// TwinCAT 3 PLC project Fraktal_Core
// Title: Fraktal_Core
// Company: fraktal-automation
// Author: fraktal-automation
// ProjectVersion: 0.25.0.0
// Description: Fraktal Core framework library: contracts, base classes (CM/EM/Unit), PermIntlk, profiler, connector base, recipe provider (Core 2.2).
// ProgramVersion: 3.1.4026.24
// libraries:
//   Tc2_Standard, * (Beckhoff Automation GmbH)
//   Tc2_EtherCAT, * (Beckhoff Automation GmbH)
//   Tc2_System, * (Beckhoff Automation GmbH)
//   Tc2_Utilities, * (Beckhoff Automation GmbH)
//   Tc3_Module, * (Beckhoff Automation GmbH)
//   Tc3_IPCDiag, * (Beckhoff Automation GmbH)
// project tree:
//   Connectivity/ FB_LineDataV3.TcPOU, FB_ShiftSchedule.TcPOU, FB_ConfigSnapshot.TcPOU, F_AppendTopologyConfig.TcPOU, FB_AsciiLink.TcPOU, FB_DeviceConnectorBase.TcPOU, FB_EcBusHealth.TcPOU, FB_EcFieldbusScanner.TcPOU, FB_IoTopologyPublisher.TcPOU, FB_LocalAccessProvider.TcPOU, FB_ConfigSetDocument.TcPOU, FB_MediumConfigStore.TcPOU, FB_PersistMediumBase.TcPOU, FB_RetainPersistMedium.TcPOU, FB_LocalPartCarrier.TcPOU (not stored), FB_LocalRecipeProvider.TcPOU, FB_LocalConfigStore.TcPOU, FB_PersistentDataWriter.TcPOU, FB_SimByteChannel.TcPOU (not stored), FB_TcpChannelTc3.TcPOU (not stored), FB_LineData.TcPOU, FB_LineLocalSource.TcPOU, FB_LineAdsSource.TcPOU
//   DUTs/ ST_ShiftRecordV3.TcDUT, ST_ShiftCalendarV3.TcDUT, ST_ShiftRowV3.TcDUT, ST_ShiftCalendarV2.TcDUT, ST_ShiftRowV2.TcDUT, ST_ConfigFeatures.TcDUT, ST_LocalRecipeCatalog.TcDUT, ST_LocalRecipeRecord.TcDUT, E_AccessLevel.TcDUT (not stored), E_AlarmState.TcDUT (not stored), E_AsciiLinkEvent.TcDUT, E_ByteChannelState.TcDUT (not stored), E_CarrierKind.TcDUT (not stored), E_Category.TcDUT (not stored), E_ChannelDir.TcDUT (not stored), E_ChannelKind.TcDUT (not stored), E_ExecState.TcDUT (not stored), E_FieldbusLossReaction.TcDUT (not stored), E_GatedAction.TcDUT, E_HbResult.TcDUT (not stored), E_HostEventKind.TcDUT, E_LinkReaction.TcDUT (not stored), E_MachineState.TcDUT (not stored), E_Mode.TcDUT (not stored), E_ModeSwitchShield.TcDUT (not stored), E_PowerGroupKind.TcDUT (not stored), E_PowerState.TcDUT (not stored), E_SafetyDeviceKind.TcDUT (not stored), E_SafetyState.TcDUT (not stored), E_ModeSwitchStyle.TcDUT (not stored), E_ModuleType.TcDUT (not stored), E_NodeState.TcDUT (not stored), E_Reason.TcDUT, E_RecipeSource.TcDUT (not stored), E_ReleaseKind.TcDUT (not stored), E_ResetClass.TcDUT (not stored), E_RunStyle.TcDUT (not stored), E_Severity.TcDUT (not stored), E_StepResult.TcDUT (not stored), E_TimeClass.TcDUT (not stored), E_Verdict.TcDUT (not stored), ST_AccessPolicy.TcDUT, ST_AlarmEvent.TcDUT, ST_AlarmMeta.TcDUT, ST_BusNode.TcDUT, ST_CommandInfo.TcDUT, E_CommandStyle.TcDUT, ST_ManualEnableStatus.TcDUT, ST_CondRecord.TcDUT (not stored), ST_CycleProfile.TcDUT, ST_CycleSummary.TcDUT, ST_DecisionRequest.TcDUT (not stored), ST_Diagnostic.TcDUT, ST_EngineeringGate.TcDUT, ST_FieldbusTopology.TcDUT, E_HmiRequestKind.TcDUT, E_ConfigKind.TcDUT, E_ConfigRestorePolicy.TcDUT, E_ConfigStore.TcDUT, E_ConfigValueType.TcDUT, E_EngUnit.TcDUT, ST_ConfigPersistStatus.TcDUT, ST_ConfigRecord.TcDUT, ST_ConfigSetInfo.TcDUT, ST_HmiRequest.TcDUT (not stored), E_ConfigStorage.TcDUT, E_LineRole.TcDUT, ST_LineDataParCfg.TcDUT, ST_LineDataParCmd.TcDUT, ST_LineDataOutCmd.TcDUT, ST_ShiftCalendar.TcDUT, ST_ShiftRecord.TcDUT, ST_LineRecord.TcDUT, ST_LineImage.TcDUT, ST_LineStatus.TcDUT, ST_ConfigAccess.TcDUT, ST_DataClassPolicy.TcDUT, ST_ConfigWriteDef.TcDUT, ST_ConfigEntry.TcDUT, ST_ConfigPage.TcDUT (not stored), ST_HmiResponse.TcDUT, ST_HostEvent.TcDUT, ST_IntlkCond.TcDUT (not stored), ST_IoChannel.TcDUT, ST_IoPointIdentity.TcDUT (not stored), ST_MeasRecord.TcDUT (not stored), ST_ModePolicy.TcDUT (not stored), ST_ModelField.TcDUT (not stored), ST_ModelId.TcDUT (not stored), ST_ModuleStatus.TcDUT, ST_ControlDomainStatus.TcDUT (not stored), ST_ControlPowerStatus.TcDUT (not stored), ST_PowerGroupStatus.TcDUT (not stored), ST_SafetyDeviceStatus.TcDUT (not stored), ST_SafetyStatus.TcDUT (not stored), ST_ModuleTiming.TcDUT (not stored), ST_Nameplate.TcDUT (not stored), ST_Oee.TcDUT (not stored), ST_OeeSample.TcDUT (not stored), ST_PartContext.TcDUT (not stored), ST_PartResult.TcDUT, ST_ReleaseReason.TcDUT (not stored), ST_ReleaseReport.TcDUT (not stored), ST_StepRecord.TcDUT, ST_StateFlag.TcDUT, ST_SequenceStepDef.TcDUT, ST_SequenceCursor.TcDUT, ST_SequenceAnnotation.TcDUT, ST_SequenceStep.TcDUT, ST_StepTiming.TcDUT, ST_SignalTowerOut.TcDUT, ST_SignalTowerParCfg.TcDUT, ST_SystemHealthInput.TcDUT, ST_SystemHealthParCfg.TcDUT, ST_SystemHealthStatus.TcDUT, ST_TimeQuality.TcDUT, ST_TimingRow.TcDUT, ST_UserRecord.TcDUT, ST_AccessImageV1.TcDUT, ST_PersistResult.TcDUT, ST_RetainDocument.TcDUT, ST_TcpVisionParCfg.TcDUT (not stored), ST_TcpVisionParCmd.TcDUT (not stored), ST_TcpVisionOutCmd.TcDUT (not stored), ST_TcpVisionOutImm.TcDUT, ST_TcpCodeReaderParCfg.TcDUT (not stored), ST_TcpCodeReaderParCmd.TcDUT (not stored), ST_TcpCodeReaderOutCmd.TcDUT (not stored), ST_TcpCodeReaderOutImm.TcDUT, ST_TcWindowsClockSampleV1.TcDUT
//   Interfaces/ I_RecipeCatalog.TcIO, I_LineSource.TcIO, I_AccessProvider.TcIO, I_AccessStore.TcIO, I_ByteChannel.TcIO (not stored), I_ControlModule.TcIO (not stored), I_DeviceConnector.TcIO (not stored), I_EquipmentModule.TcIO (not stored), I_EventSink.TcIO (not stored), I_HostEventSink.TcIO, I_FieldbusScanner.TcIO, I_ConfigSource.TcIO, I_ConfigPersistence.TcIO, I_ConfigStore.TcIO, I_PersistMedium.TcIO, I_ManualTarget.TcIO, I_Module.TcIO, I_PartCarrier.TcIO (not stored), I_Sequence.TcIO, I_SequenceHost.TcIO, I_RecipeStore.TcIO, I_RecipeProvider.TcIO, I_Unit.TcIO (not stored), I_VerdictProvider.TcIO (not stored)
//   BaseClasses/ FB_AccessManager.TcPOU, FB_AlarmLog.TcPOU, FB_AsciiDeviceCM.TcPOU, FB_EngineeringMode.TcPOU, FB_ConfigPager.TcPOU, FB_ModuleBase.TcPOU, FB_ControlModuleBase.TcPOU (not stored), FB_CycleProfiler.TcPOU, FB_SignalTower.TcPOU, FB_SystemHealthPublisher.TcPOU, FB_CompositeModuleBase.TcPOU, FB_EquipmentModuleBase.TcPOU (not stored), FB_HostEventPublisher.TcPOU, FB_SequenceBase.TcPOU, FB_UnitBase.TcPOU
//   Platform/ F_ReasonMeta.TcPOU, F_ReasonMetaByIndex.TcPOU, F_RationalizeDiagnostic.TcPOU, F_Sha256.TcPOU, F_Crc32.TcPOU, F_ValidPersistKey.TcPOU, FB_FilePersistMedium.TcPOU, FB_TcIpcDiagnostics.TcPOU, F_Now.TcPOU (not stored), FB_ConfigSetJson.TcPOU, F_ManualEnable.TcPOU, F_TryParseNumber.TcPOU, F_EngUnitSymbol.TcPOU, F_TimeSynchronized.TcPOU, FB_TcSystemHealthProbe.TcPOU, F_TcWindowsClockCrc.TcPOU, FB_TcWindowsTime.TcPOU, F_TimingUpdate.TcPOU (not stored)
//   DeviceCMs/ FB_TcpCodeReaderCM.TcPOU, FB_TcpVisionCM.TcPOU
//   Params/ PL_Fraktal.TcGVL, PL_FraktalCompat.TcGVL, PL_FraktalEngineering.TcGVL, PL_ReasonCatalog.TcGVL, PL_TcpDevReasons.TcGVL (not stored)
//   GVLs/ GVL_FraktalTime.TcGVL
//   PermIntlk/ FB_PermIntlk.TcPOU
// real-time tasks:
//   TASK PlcTask: cycle T#10ms, priority 20, ADS port 350

// ---- DUTs/ST_ShiftRecordV3.TcDUT
// Core §8.5.2(b) - one closed shift, exactly as its figures stood at the boundary.
TYPE ST_ShiftRecordV3 :
STRUCT
    SchemaVersion : UINT := 3;
    ProductionTarget : UDINT;
    ShiftIndex       : INT;     // 1..MAX_SHIFTS
    StartAt          : DT;      // §2.7 clock (UTC)
    EndAt            : DT;
    TimeSynchronized : BOOL;    // FALSE if either boundary was crossed on an unsynchronized clock
    ManualReset      : BOOL;    // counts or OEE were reset by hand during this shift
    GoodCount        : UDINT;
    NokCount         : UDINT;
    ReworkCount      : UDINT;
    RunMs            : UDINT;
    DownMs           : UDINT;
    IdleMs           : UDINT;
    Availability     : REAL;    AvailValid : BOOL;
    Performance      : REAL;    PerfValid  : BOOL;
    Quality          : REAL;    QualValid  : BOOL;
    Oee              : REAL;    OeeValid   : BOOL;
END_STRUCT
END_TYPE

// ---- DUTs/ST_ShiftCalendarV3.TcDUT
TYPE ST_ShiftCalendarV3 :
STRUCT
    SchemaVersion : UINT;
    UtcOffsetMin : DINT;
    Rows : ARRAY[1..PL_Fraktal.MAX_WEEKLY_SHIFTS] OF ST_ShiftRowV3;
END_STRUCT
END_TYPE

// ---- DUTs/ST_ShiftRowV3.TcDUT
TYPE ST_ShiftRowV3 :
STRUCT
    StartMin : DINT := -1;
    DurationMin : DINT := 1440;
    ActiveDays : DINT;
    ProductionTarget : DINT;
END_STRUCT
END_TYPE

// ---- DUTs/ST_ShiftCalendarV2.TcDUT
TYPE ST_ShiftCalendarV2 :
STRUCT
    SchemaVersion : UINT;
    UtcOffsetMin : DINT;
    Rows : ARRAY[1..PL_Fraktal.MAX_SHIFTS] OF ST_ShiftRowV2;
END_STRUCT
END_TYPE

// ---- DUTs/ST_ShiftRowV2.TcDUT
TYPE ST_ShiftRowV2 :
STRUCT
    StartMin : DINT := -1;
    DurationMin : DINT := 1440;
    ActiveDays : DINT;
END_STRUCT
END_TYPE

// ---- DUTs/ST_ConfigFeatures.TcDUT
TYPE ST_ConfigFeatures :
STRUCT
    ExportCurrentConfig : BOOL;
END_STRUCT
END_TYPE

// ---- DUTs/ST_LocalRecipeCatalog.TcDUT
// TC3 retained catalog image, separate from the volatile seed pointer registry.
TYPE ST_LocalRecipeCatalog :
STRUCT
    SchemaVersion : UINT;
    Count : INT;
    Records : ARRAY[1..PL_Fraktal.MAX_RECIPES] OF ST_LocalRecipeRecord;
END_STRUCT
END_TYPE

// ---- DUTs/ST_LocalRecipeRecord.TcDUT
// Provider-owned, pointer-free retained recipe storage. Data begins with its own schema.
TYPE ST_LocalRecipeRecord :
STRUCT
    SchemaVersion : UINT := 1;
    ModelCode : STRING(64);
    RecipeKey : STRING(80);
    DataSize : UDINT;
    Data : ARRAY[1..PL_Fraktal.MAX_MODEL_DATA_BYTES] OF BYTE;
END_STRUCT
END_TYPE

// ---- DUTs/E_AsciiLinkEvent.TcDUT
// Core §3.15.1a - what one FB_AsciiLink tick produced. The link reports; its owner
// (a device CM, or a connector) decides what each event means for it.
{attribute 'qualified_only'}
TYPE E_AsciiLinkEvent :
(
    NONE          := 0,
    RESPONSE      := 1,   // one terminated response is in Response
    TIMEOUT       := 2,   // the outstanding request got no response in RespTimeout
    OVERFLOW      := 3,   // no terminator within the receive bound: buffer dropped
    CHANNEL_FAULT := 4,   // the transport reported FAULT; the channel was closed
    INVALID_STATE := 5    // the transport reported a state outside the contract
) DINT;
END_TYPE

// ---- DUTs/E_GatedAction.TcDUT
// Core §7.7(a) — the enumerated protected actions (array index 0..11)
{attribute 'qualified_only'}
TYPE E_GatedAction :
(
    DATA_READ     := 0,   // view ParCfg/StationCfg values
    DATA_WRITE    := 1,   // edit ParCfg/StationCfg (§3.8a)
    MANUAL        := 2,   // manual movements default (§7.6 may raise per function)
    CHANGEOVER    := 3,   // SetModel (§3.1b)
    MODE_CHANGE   := 4,   // SetMode (§3.4)
    START_STOP    := 5,
    ALARM_HISTORY := 6,   // browse §8.3 ring
    ALARM_RESET   := 7,   // OperatorReset (§8.3(b))
    ACCESS_POLICY := 8,   // editing the policy itself
    ALARM_SHELVE  := 9,   // §8.10 shelve/unshelve an annunciated alarm
    POWER_CONTROL := 10,  // §9.8 Control On/Off and power-group requests
    CONFIG_SET    := 11   // §3.8b save/load/import a whole parameter set
) DINT;
END_TYPE

// ---- DUTs/E_HostEventKind.TcDUT
// Core §11.6.1 — fixed, append-only L3/MES event vocabulary.
{attribute 'qualified_only'}
TYPE E_HostEventKind :
(
    NONE := 0,
    PART_RECEIVED := 1,
    PROCESSING_STARTED := 2,
    PROCESSED := 3,
    PROCESSING_ABORTED := 4,
    CHANGEOVER_STARTED := 5,
    CHANGEOVER_DONE := 6,
    TOOL_CHANGED := 7,
    MATERIAL_CHANGED := 8,
    MODE_CHANGED := 9,
    NOK := 10
) DINT;
END_TYPE

// ---- DUTs/E_Reason.TcDUT
// Core §8.8 — reason-code vocabulary. Framework bands only; module TYPES declare
// their band codes (10000+) as DINT constants in their own library and assign them
// to E_Reason members of ST_Diagnostic (enum is deliberately NOT 'strict' so band
// codes outside this declaration remain assignable — see IMPLEMENTATION_NOTES §3).
// Registry: Core §8.8. Codes are positive (PLCopen ErrorID is unsigned).
{attribute 'qualified_only'}
TYPE E_Reason :
(
    NONE                    := 0,

    // ── System 10–21: controller & clock health (Core §8.12, §2.7) ──
    TASK_OVERRUN            := 10,
    TASK_JITTER_HIGH        := 11,
    CPU_LOAD_HIGH           := 12,
    MEMORY_LOW              := 13,
    IPC_TEMP_HIGH           := 14,
    FIELDBUS_MASTER_FAULT   := 15,
    DC_SYNC_LOST            := 16,
    TIME_SYNC_LOST          := 17,
    UTILITY_DEVIATION       := 18,
    IPC_FAN_FAULT           := 19,
    STORAGE_HEALTH_LOW      := 20,
    CONTROLLER_METRICS_UNAVAILABLE := 21,

    // ── Framework 2000–2009: common flow reasons (Core §8.8) ──
    TIMEOUT                 := 2001,
    PERMISSIVE_NOT_MET      := 2002,
    INTERLOCK_DROPPED       := 2003,
    RECIPE_INVALID          := 2004,
    STEP_STALLED            := 2005,
    RETRY_EXHAUSTED         := 2006,
    CYCLE_TIME_DEGRADED     := 2007,   // maintenance event on timing drift (Core §8.11.4(d)/§8.12)
    UNSUPPORTED_COMMAND     := 2008,   // command outside the type's supported set (§5.6)

    // ── Framework 2010–2019: external device / link supervision (Core §3.15) ──
    LINK_TIMEOUT            := 2010,
    DEVICE_NOT_READY        := 2011,
    DEVICE_PROTOCOL_ERROR   := 2012,

    // ── Framework 2020–2029: traceability / part context (Core §3.16) ──
    CARRIER_READ_FAILED     := 2020,
    CARRIER_WRITE_FAILED    := 2021,
    PART_ID_MISMATCH        := 2022,
    RESULT_RECORD_REJECTED  := 2023,
    // §3.16.3 canonical part-lifecycle events (MESSAGE ring entries, not faults)
    EVENT_PART_RECEIVED           := 2024,
    EVENT_PART_PROCESSING_STARTED := 2025,
    EVENT_PART_PROCESSED          := 2026,
    EVENT_PART_PROCESSING_ABORTED := 2027,

    // ── Framework 2030–2039: engineering / commissioning build gates (Core §7.5) ──
    // One LOW/SYSTEM event per ACTIVE gate: not clearable, not shelvable, and
    // AUTO_RESET so it never blocks the commissioning it exists to serve.
    COMMISSIONING_GATE_ACTIVE := 2030,

    // ── Framework 2040–2049: configuration persistence & parameter sets (§3.8b) ──
    // A retained image was REJECTED (an unrecognized schema version), so the
    // owning module is running on its declared defaults. Version 0 — never
    // written — is a first boot that lost nothing and raises nothing.
    CONFIG_RESTORE_LOST     := 2040,
    // An accepted write did not reach non-volatile storage inside the declared
    // window. Transport ack and Accepted mean LIVE, never DURABLE.
    CONFIG_PERSIST_FAILED   := 2041,
    // A parameter-set load was refused. Staged and all-or-nothing: nothing in
    // the machine changed, and the refusal names the offending (Scope, WriteKey).
    CONFIG_SET_REJECTED     := 2042,
    // §8.3 audit trail for a set that WAS applied — an event, not an alarm.
    EVENT_CONFIG_SET_APPLIED := 2043,

    // ── Framework 2900–2909: framework self-test (never raised in production) ──
    TEST_FAULT              := 2901
) DINT;
END_TYPE

// ---- DUTs/ST_AccessPolicy.TcDUT
// Core §7.7(b) — per-station required level per action. SHIPPED DEFAULT: fully open
// (NONE everywhere) — locking down is a deliberate deployment decision, reviewed at
// commissioning (§14). Held as persistent station configuration (§3.8a).
TYPE ST_AccessPolicy :
STRUCT
    Required       : ARRAY[0..11] OF E_AccessLevel;  // index = TO_INT(E_GatedAction)
    SessionTimeout : TIME := T#0S;                   // idle auto-logout; T#0S = never
END_STRUCT
END_TYPE

// ---- DUTs/ST_AlarmEvent.TcDUT
// Core §8.3(a) — one alarm/event with full lifecycle. Same reason vocabulary as
// every diagnostic (§8.8): the event IS the diagnostic plus lifecycle.
TYPE ST_AlarmEvent :
STRUCT
    ReasonCode  : E_Reason;
    Description : STRING(255);
    SourcePath  : STRING(255);   // module browse path (§4.8) = historian tag path
    IoTag       : STRING(80);    // exact implicated electrical tag; untranslated
    IoAddress   : STRING(80);    // terminal/channel locator
    Severity    : E_Severity;
    Category    : E_Category;
    ResetClass  : E_ResetClass;
    State       : E_AlarmState;
    ComeAt      : DT;            // synchronized stamps (§2.7)
    GoneAt      : DT;
    ResetAt     : DT;            // MANUAL_RESET only
    Duration    : TIME;          // monotonic come->gone (§8.11.4(e) two-clock rule)
    Shelved     : BOOL;          // §8.10 annunciation suppressed (control unaffected)
    ShelvedUntil: DT;            // display only; enforcement is the log's countdown
    ComeTimeSynchronized : BOOL;
    GoneTimeSynchronized : BOOL;
    ResetTimeSynchronized : BOOL;
    ShelfTimeSynchronized : BOOL;
END_STRUCT
END_TYPE

// ---- DUTs/ST_AlarmMeta.TcDUT
// Core §8.9 — runtime rationalization record for one ReasonCode: what the operator
// should DO, what happens if they don't, and whether shelving is permitted.
TYPE ST_AlarmMeta :
STRUCT
    ReasonCode     : E_Reason;
    OperatorAction : STRING(255);  // "what do I do about this?"
    Consequence    : STRING(255);
    Priority       : E_Severity;    // one reason, one priority everywhere
    Category       : E_Category;    // PROCESS / SAFETY / SYSTEM
    Shelvable      : BOOL;         // §8.10: no record or FALSE -> not shelvable
END_STRUCT
END_TYPE

// ---- DUTs/ST_BusNode.TcDUT
// Core §10.5.1 — one fieldbus node. The node/channel arrays are populated at
// runtime from the master's diagnostics (TC3 §10.6: EtherCAT/ADS); this is the
// published shape the generic HMI renders. Children are referenced by index into
// the master's flat node table to keep the DUT bounded (no recursion in IEC types).
TYPE ST_BusNode :
STRUCT
    // §3.10.2 — identity/topology members are activation-static: excluded from
    // the cyclic OPC UA tree and served via the root Unit's config manifest
    // (F_AppendTopologyConfig). Only live state stays cyclically published.
    {attribute 'OPC.UA.DA' := '0'}
    Name        : STRING(80);
    {attribute 'OPC.UA.DA' := '0'}
    DescriptionKey : STRING(160); // hardware-description localization key
    {attribute 'OPC.UA.DA' := '0'}
    TypeId      : STRING(80);   // vendor/product
    {attribute 'OPC.UA.DA' := '0'}
    Address     : STRING(40);   // topological + logical
    State       : E_NodeState;
    LinkOk      : BOOL;
    {attribute 'OPC.UA.DA' := '0'}
    ParentIdx   : INT;          // index of parent node in the flat table (0 = root)
    {attribute 'OPC.UA.DA' := '0'}
    ChannelCount: INT;
    Channels    : ARRAY[1..PL_Fraktal.MAX_NODE_CHANNELS] OF ST_IoChannel;
END_STRUCT
END_TYPE

// ---- DUTs/ST_CommandInfo.TcDUT
// Core §7.6.1 — one entry in a module's self-describing command catalog.
// Value is what ExecuteCommand accepts (§3.2); Label is the button text.
TYPE ST_CommandInfo :
STRUCT
    Value : DINT;
    Label : STRING(120);   // localization key; resolved by the HMI catalog
    // §7.6.1 - ONESHOT (default) goes to ExecuteCommand; HELD is re-asserted
    // every scan through RequestHeldCommand and stops when the asking stops.
    // Additive with a zero default, so a consumer that predates it reads
    // every existing entry as ONESHOT, which is what they all were (§1.5).
    Style : E_CommandStyle;
END_STRUCT
END_TYPE

// ---- DUTs/E_CommandStyle.TcDUT
// Core §7.6.1 - how a published command is OPERATED, so a generic HMI can render
// it without knowing the module type (O1: no per-type HMI code).
//
// ONESHOT is the ordinary PLCopen command: press once, the module runs it to
// Done. HELD is a command that only acts while the operator keeps asking - a
// jog. The distinction is not cosmetic: a held action is re-asserted every scan
// and STOPS when the asking stops, including when it stops because the network
// stalled rather than because the operator let go (O10).
{attribute 'qualified_only'}
TYPE E_CommandStyle : (ONESHOT := 0, HELD := 1) DINT;
END_TYPE

// ---- DUTs/ST_ManualEnableStatus.TcDUT
// Core §9 — "is a safety-rated enabling device permitting manual motion right
// now?", derived from the §9 device rows and never authored.
//
// This is STATUS, not authority. §9 is read-only to the application and the PLC
// never infers "safe" from it: the safety system decides whether guards may be
// open, enforces the reduced speed, and mutes the interlock. What this record
// says is only what the certified system has already published about its
// enabling device — so that a release (§7.6) can be written against a fact with
// a provenance, instead of against a boolean a station assembled from standard
// I/O.
//
// A three-position enabling device reads as permitting ONLY in its middle
// position. Released and panic-squeezed are both non-permitting, which is the
// entire reason the device has three positions rather than two.
TYPE ST_ManualEnableStatus :
STRUCT
    Present    : BOOL;          // at least one enabling device is mirrored here
    Held       : BOOL;          // one is permitting NOW - safety-evaluated, standard PLC cannot set
    DeviceName : STRING(80);    // which one, so a release report can name it (§7.6.0)
END_STRUCT
END_TYPE

// ---- DUTs/ST_CycleProfile.TcDUT
// Core §8.11.4(b)/(f) — one completed cycle: ordered waterfall + time-class split.
// ByClass is indexed by TO_INT(E_TimeClass): 0=WORK 1=WAIT_UPSTREAM 2=WAIT_DOWNSTREAM
// 3=WAIT_OPERATOR 4=WAIT_EXTERNAL.
TYPE ST_CycleProfile :
STRUCT
    CycleNo   : UDINT;
    Started   : DT;
    StartedTimeSynchronized : BOOL;
    Total     : TIME;     // reconciles with the §8.11.1 CycleTime
    WorkTime  : TIME;     // §8.11.4(f): THE REAL CYCLE TIME (= ByClass[WORK])
    WaitTime  : TIME;     // Total - WorkTime (all wait classes)
    ByClass   : ARRAY[0..4] OF TIME;
    NSteps    : INT;
    Truncated : BOOL;     // more step changes than MAX_PROFILE_STEPS
    Steps     : ARRAY[1..PL_Fraktal.MAX_PROFILE_STEPS] OF ST_StepTiming;
END_STRUCT
END_TYPE

// ---- DUTs/ST_CycleSummary.TcDUT
// Core §8.11.4 — one completed cycle's totals for the trend ring: enough to chart
// WHY cycle time moved (work vs each wait class) without the full step waterfall.
TYPE ST_CycleSummary :
STRUCT
    CycleNo  : UDINT;
    Started  : DT;                    // synchronized wall clock (Core §2.7)
    StartedTimeSynchronized : BOOL;
    Total    : TIME;
    WorkTime : TIME;                  // §8.11.4(f) — the real cycle time
    WaitTime : TIME;
    ByClass  : ARRAY[0..4] OF TIME;   // indexed by TO_INT(E_TimeClass)
END_STRUCT
END_TYPE

// ---- DUTs/ST_Diagnostic.TcDUT
// Core §8.8 — the full first-out reason record
TYPE ST_Diagnostic :
STRUCT
    ReasonCode  : E_Reason;      // named reason; ErrorID = TO_DWORD(ReasonCode)
    SourcePath  : STRING(255);   // OPC UA browse path of the module/condition (Core §4.8)
    Description : STRING(255);   // localization key (from PermIntlk or module); never operator prose
    IoTag       : STRING(80);    // untranslated schematic/electrical tag of implicated channel
    IoAddress   : STRING(80);    // terminal/channel locator, e.g. EL1809 Ch5
    Severity    : E_Severity;    // LOW | MED | HIGH (Core §8.1)
    Category    : E_Category;    // PROCESS | SAFETY | SYSTEM
    Since       : DT;            // first-out timestamp (synchronized clock, Core §2.7)
    TimeSynchronized : BOOL;      // FALSE when the selected source is unavailable/out of tolerance
END_STRUCT
END_TYPE

// ---- DUTs/ST_EngineeringGate.TcDUT
// Core §7.5.1 — one ACTIVE commissioning/engineering gate in the station register.
// There is deliberately no `Active` member: a gate is a build constant (§7.5.1),
// so an inactive gate is not registered at all. A production station therefore
// publishes an EMPTY register, and the surfaces its gates control are invisible
// rather than merely disabled (§3.9).
TYPE ST_EngineeringGate :
STRUCT
    Name           : STRING(80);    // stable gate identity, e.g. 'OUTPUT_FORCING'
    DescriptionKey : STRING(160);   // localization key for the §7.5.2 annunciation
END_STRUCT
END_TYPE

// ---- DUTs/ST_FieldbusTopology.TcDUT
// Core §10.5.1 — bounded published fieldbus table plus mapping validation.
// Physical discovery fills nodes; the project catalog joins approved I/O metadata.
TYPE ST_FieldbusTopology :
STRUCT
    NodeCount : INT;
    Nodes : ARRAY[1..PL_Fraktal.MAX_BUS_NODES] OF ST_BusNode;
    MappingValid : BOOL;
    MappingDiagnostic : STRING(255); // localization key; empty when valid
    // §10.5.1 rule 3 - are held force set-points currently applied? This lives
    // in the PUBLISHED table rather than in one FB_IoTopologyPublisher instance
    // because a project attaches several to the same data (the catalog defines
    // channel identity, the hardware driver moves live values), and two copies
    // of this flag would let them disagree about whether a force is live.
    {attribute 'OPC.UA.DA' := '0'}
    ForcesEnabled : BOOL;
END_STRUCT
END_TYPE

// ---- DUTs/E_HmiRequestKind.TcDUT
// Core §3.10/§14 — generic OPC UA request mailbox operation.
// Append-only: ordinal values are a transport contract with every HMI adapter.
{attribute 'qualified_only'}
TYPE E_HmiRequestKind :
(
    NONE             := 0,
    LOGIN            := 1,
    LOGOUT           := 2,
    SET_MODE         := 3,
    SET_MODEL        := 4,
    START            := 5,
    STOP             := 6,
    CONTROL_ON       := 7,
    CONTROL_OFF      := 8,
    OPERATOR_RESET   := 9,
    DECISION_ANSWER  := 10,
    MANUAL_COMMAND   := 11,
    SET_RUN_STYLE    := 12,
    STEP_REQUEST     := 13,
    SET_HOLD_RUN     := 14,
    RELEASE_START    := 15,
    RELEASE_MANUAL   := 16,
    RELEASE_ACTION   := 17,
    RESET_OEE        := 18,
    WRITE_CONFIG     := 19,
    SHELVE_ALARM     := 20,
    UNSHELVE_ALARM   := 21,
    FORCE_CHANNEL    := 22,
    QUERY_CONFIG     := 23,   // §3.10.2 config-manifest page request (IntValue = page)
    SET_ACCESS_LEVEL := 24,   // §7.7 policy: IntValue=gate, TextValue=level ordinal
    SET_SESSION_TIMEOUT := 25, // §7.7 policy: DurationMs, 0 = never
    LAMP_TEST        := 26,    // §8.13 bounded signal-tower test
    // §3.8c — a capture is a write whose value comes from the machine. The root
    // already owned CaptureConfig; without a request kind no client could reach
    // it, and §3.8c(a) requires a capture to be routed through this same
    // acknowledged mailbox. TargetPath=Scope, NameValue=WriteKey, IntValue=rev.
    CAPTURE_CONFIG   := 27,
    // §3.8b parameter sets. TextValue = set name; IntValue = E_ConfigKind for a
    // save (which class of records the set carries). All three are CONFIG_SET,
    // separately from the DATA_WRITE that edits one value.
    SAVE_CONFIG_SET  := 28,
    LOAD_CONFIG_SET  := 29,
    LIST_CONFIG_SETS := 30,
    // §3.8b — an ENGINEER-level operator accepts a restore loss. Under
    // BLOCK_UNTIL_ACKNOWLEDGED this is what releases START_STOP again.
    ACK_CONFIG_RESTORE := 31,
    // §3.8b — move a set as TEXT. Export serves one JSON line per request
    // (IntValue = line; 0 = header), import takes one back (TextValue = the line,
    // BoolValue = this is the last one). Paged for the same reason QUERY_CONFIG
    // is: no full set document ever has to exist in PLC memory. A line longer
    // than TextValue travels in pieces: IntValue = 1 holds a piece, the next
    // request without it completes the line (additive; an older root refuses a
    // piece as an unreadable line, so it fails closed).
    EXPORT_CONFIG_SET := 32,
    IMPORT_CONFIG_SET := 33,
    // §7.6.1a hold-to-run. TargetPath = module, IntValue = command value,
    // BoolValue = TRUE while the operator holds it. The client REFRESHES this
    // while held; the root drops the hold on its own if refreshes stop, so a
    // closed HMI or a dead link stops the motion rather than latching it.
    MANUAL_HELD := 34,
    // §3.8b - remove one named set (TextValue = set name). CONFIG_SET, like the
    // other set operations. Without it a store that has held MAX_CONFIG_SETS
    // names could only ever overwrite one of them again.
    DELETE_CONFIG_SET := 35,
    // §3.8d - edit a data class's level. NameValue = ClassId, IntValue =
    // E_AccessLevel ordinal, BoolValue = TRUE for the write level. ACCESS_POLICY.
    SET_CLASS_LEVEL := 36,
    // Optional bounded catalog: inactive clone; NameValue = new code,
    // IntValue = source model (0 running), BoolValue = from saved Model set,
    // TextValue = source set name. Only offered with positive ModelCapacity.
    CREATE_MODEL := 37,
    // Read-only snapshot export, TextValue = export name, IntValue = CfgKind,
    // DurationMs = model index (0 running). Header returned as line zero;
    // EXPORT_CONFIG_SET continues the immutable connection-local document.
    EXPORT_CURRENT_CONFIG := 38
) DINT;
END_TYPE

// ---- DUTs/E_ConfigKind.TcDUT
// Core §3.8a/§3.10.2 — persistent configuration ownership class.
// Ordinals are an append-only PLC/HMI transport contract.
{attribute 'qualified_only'}
TYPE E_ConfigKind :
(
    PAR_CFG     := 0,
    STATION_CFG := 1,
    LINE_CFG    := 2      // §3.8e shared by every station on a line; one owner
) DINT;
END_TYPE

// ---- DUTs/E_ConfigRestorePolicy.TcDUT
// Core §3.8b — what a station DOES about a configuration image it could not
// restore. The loss itself is never silent either way; this chooses the
// consequence, and the deployment declares it rather than inheriting a habit.
// Ordinals are an append-only PLC/HMI transport contract.
{attribute 'qualified_only'}
TYPE E_ConfigRestorePolicy :
(
    // Shipped default: the station runs on its declared defaults and the
    // annunciation stands until an operator acknowledges it. A machine that
    // still moves is the right answer for a station whose lost values are
    // conveniences; the standing alarm is what stops it being silent.
    DEFAULTS_AND_ANNUNCIATE  := 0,
    // No START_STOP release until an operator of at least ENGINEER level
    // acknowledges the loss. For a station whose commissioned values are the
    // difference between a good part and a wrecked tool, running on defaults
    // while presenting itself as commissioned is the failure to prevent.
    BLOCK_UNTIL_ACKNOWLEDGED := 1
) DINT;
END_TYPE

// ---- DUTs/E_ConfigStore.TcDUT
// Core §3.8b — the medium behind an I_ConfigStore implementation, published so
// an operator can see WHERE this station's parameter sets actually live before
// trusting that a save survived. The store moves records and nothing else: it
// does not validate, does not know what a value means, and is never an
// authorization authority (§5.6, §14).
// Ordinals are an append-only PLC/HMI transport contract.
{attribute 'qualified_only'}
TYPE E_ConfigStore :
(
    LOCAL_RETAIN := 0,   // in-PLC retentive memory (FB_LocalConfigStore, the shipped default)
    FILE_JSON    := 1,   // controller/host file system, serialized set document
    FILE_XML     := 2,
    EXTERNAL     := 3    // database, asset system or MES behind a §3.15 connector
) DINT;
END_TYPE

// ---- DUTs/E_ConfigValueType.TcDUT
// Core §3.8a/§3.10.2 — configuration value representation accepted by the
// owning typed write handler. Ordinals mirror the generic HMI CfgType enum.
// Append new values only.
{attribute 'qualified_only'}
TYPE E_ConfigValueType :
(
    NUMBER  := 0,
    TEXT    := 1,
    BOOLEAN := 2,
    DURATION := 3   // TwinCAT binding name for Core TIME; TIME is a reserved keyword
) DINT;
END_TYPE

// ---- DUTs/E_EngUnit.TcDUT
// Core §3.10.2 - the engineering unit of a configuration value, as a CODE.
// A unit is a vocabulary entry like any other text the operator reads: the PLC
// publishes the code and the HMI owns the symbol, translated with everything
// else (std.unit.<name>). NONE = 0 = the value has no unit, and the HMI then
// shows none. Ordinals are the HMI contract (lib/domain/types.dart EngUnit,
// lint rule E1) - append only.
{attribute 'qualified_only'}
TYPE E_EngUnit :
(
    NONE                          := 0,
    MILLISECOND                   := 1,
    SECOND                        := 2,
    MINUTE                        := 3,
    HOUR                          := 4,
    MICROMETER                    := 5,
    MILLIMETER                    := 6,
    METER                         := 7,
    DEGREE                        := 8,
    MILLIMETER_PER_SECOND         := 9,
    METER_PER_MINUTE              := 10,
    DEGREE_PER_SECOND             := 11,
    MILLIMETER_PER_SECOND_SQUARED := 12,
    BAR                           := 13,
    KILOPASCAL                    := 14,
    NEWTON                        := 15,
    KILONEWTON                    := 16,
    NEWTON_METER                  := 17,
    GRAM                          := 18,
    KILOGRAM                      := 19,
    DEGREE_CELSIUS                := 20,
    PERCENT                       := 21,
    REVOLUTION_PER_MINUTE         := 22,
    HERTZ                         := 23,
    VOLT                          := 24,
    AMPERE                        := 25,
    WATT                          := 26,
    KILOWATT                      := 27,
    LITER                         := 28,
    LITER_PER_MINUTE              := 29,
    PIECE                         := 30,
    PIECE_PER_MINUTE              := 31,
    PIECE_PER_HOUR                := 32
) DINT;
END_TYPE

// ---- DUTs/ST_ConfigPersistStatus.TcDUT
// Core §3.8b — the root's published answer to "is my configuration actually
// safe?". Transport acknowledgement and Accepted (§3.10(a″)) mean a value is
// LIVE; they say nothing about whether it is DURABLE, and a station that cannot
// persist is a station that will silently revert at its next restart. That has
// to be visible BEFORE the restart rather than discovered after it, which is
// what this record exists for.
TYPE ST_ConfigPersistStatus :
STRUCT
    // Durability of ordinary accepted writes.
    Pending      : BOOL;   // an accepted write has not yet reached non-volatile storage
    Failed       : BOOL;   // the store rejected it, or the declared window elapsed
    // The DECLARED bounded window a write has to become durable. Defaulted HERE
    // rather than in the root's OnInit on purpose: a composition root declares
    // its window at Setup, which runs BEFORE the first cyclic scan, and an
    // OnInit assignment would silently overwrite the declaration it was given.
    WindowMs     : UDINT := PL_Fraktal.CONFIG_PERSIST_WINDOW_MS;
    PendingSince : DT;     // when the oldest still-pending write was accepted
    StorePresent : BOOL;   // a set store is wired (save/load/list are offered)
    StoreKind    : E_ConfigStore;

    // Restore (§3.8b fail-closed startup).
    RestorePolicy       : E_ConfigRestorePolicy;
    RestoreLost         : BOOL;       // a retained image was rejected somewhere in this subtree
    RestoreAcknowledged : BOOL;       // an ENGINEER-level operator has accepted the loss
    LostPath            : STRING(80); // canonical path of the LAST module that reported one

    // Last set operation, so a refusal names the offending value rather than
    // just failing (§3.8b: one rejection aborts the load NAMING the record).
    LastSetName     : STRING(80);
    LastSetRecords  : INT;
    LastRejectScope : STRING(80);
    LastRejectKey   : STRING(160);
END_STRUCT
END_TYPE

// ---- DUTs/ST_ConfigRecord.TcDUT
// Core §3.8b — ONE value inside a parameter set, keyed by (Scope, WriteKey).
//
// This is the type that makes §3.8b's central prohibition structural. A byte
// image of a station's configuration - one aggregate memory-copied in and out -
// SHALL NOT be used, because it reinterprets retained bytes silently when a type
// changes, carries no per-value identity a file/database/MES can bind to, and
// cannot reject one bad value without rejecting all of them. A set built from
// these records has the opposite property on all three counts.
//
// Widths are not arbitrary: Scope is ST_ModuleStatus.Name, WriteKey is the
// §3.10.2 mutation identity, and ValueText is capped at the same 80 characters
// M_RegisterConfigWrite refuses to exceed for a text target - so a record can
// always carry any value the write path would have accepted.
TYPE ST_ConfigRecord :
STRUCT
    Scope     : STRING(80);    // owning module's canonical identity (= Status.Name)
    WriteKey  : STRING(160);   // §3.10.2 mutation identity, scoped to that module
    Revision  : UDINT;         // the capability revision the value was taken at
    Kind      : E_ConfigKind;
    ValueType : E_ConfigValueType;
    ValueText : STRING(80);    // serialized exactly as a WRITE_CONFIG would carry it
END_STRUCT
END_TYPE

// ---- DUTs/ST_ConfigSetInfo.TcDUT
// Core §3.8b — the header of one named parameter set: everything needed to
// decide whether this set belongs on this machine BEFORE any value changes.
//
// RootIdentity and ConfigRev are the two that matter. A set taken from another
// root, or at a revision whose capabilities have since changed meaning, is not
// a set this root can silently replay - and the difference is only visible if
// the set says where and when it came from.
TYPE ST_ConfigSetInfo :
STRUCT
    Used             : BOOL;         // slot occupied (a store publishes a bounded table)
    SetName          : STRING(80);
    RootIdentity     : STRING(80);   // canonical identity of the root that produced it
    SetSchema        : UINT;         // set-document schema version (§13)
    ConfigRev        : UDINT;        // §3.10.2 manifest revision it was taken at
    Kind             : E_ConfigKind; // STATION_CFG = station set; PAR_CFG = model set
    ModelCode        : STRING(64);   // model set only; '' for a station set
    RecordCount      : INT;
    CreatedAt        : DT;           // §2.7 synchronized clock
    TimeSynchronized : BOOL;         // quality of CreatedAt; FALSE = display as untrusted
END_STRUCT
END_TYPE

// ---- DUTs/E_ConfigStorage.TcDUT
// Core §3.8b — the PLC type actually behind a registered editable value.
// E_ConfigValueType says how the HMI renders and validates a value; this says
// how the framework parses and stores it. They are different questions: a
// settle time and a cycle count both publish as a number, and writing one into
// the other's storage would be a silent corruption rather than a rejection.
// Local to the binding (never transported), so this enum may be reordered.
{attribute 'qualified_only'}
TYPE E_ConfigStorage :
(
    NONE      := 0,   // unregistered — fails closed
    AS_BOOL   := 1,
    AS_INT    := 2,
    AS_DINT   := 3,
    AS_UDINT  := 4,
    AS_REAL   := 5,
    AS_LREAL  := 6,
    AS_TIME   := 7,   // serialized as whole milliseconds, per the HMI number contract
    AS_STRING := 8    // STRING(80)
) DINT;
END_TYPE

// ---- DUTs/E_LineRole.TcDUT
// Core §3.8e - which copy of a line's data this controller holds.
{attribute 'qualified_only'}
TYPE E_LineRole :
(
    NONE   := 0,   // not set up
    OWNER  := 1,   // the one authoritative, editable copy
    MIRROR := 2    // a read-only copy applied whole from the owner
) DINT;
END_TYPE

// ---- DUTs/ST_LineDataParCfg.TcDUT
TYPE ST_LineDataParCfg :
STRUCT
    SchemaVersion : UINT := 1;  // §3.8: first member
    StaleAfterMs  : UDINT;       // mirror: declared window for staying current (§3.8e(d))
END_STRUCT
END_TYPE

// ---- DUTs/ST_LineDataParCmd.TcDUT
TYPE ST_LineDataParCmd :
STRUCT
    Reserved : BOOL; // line data takes no command: physical four-structure contract
END_STRUCT
END_TYPE

// ---- DUTs/ST_LineDataOutCmd.TcDUT
TYPE ST_LineDataOutCmd :
STRUCT
    Reserved : BOOL; // no command result
END_STRUCT
END_TYPE

// ---- DUTs/ST_ShiftCalendar.TcDUT
// Core §8.5.2(a) - a line's shift calendar. Line data (§3.8e): edited once at the
// owner, mirrored whole. Compact on purpose - five registered values - so a line
// module keeps room for the project's own line data. A shift is named by its index
// ('Shift 1'), which the front end localizes; no operator text lives here.
TYPE ST_ShiftCalendar :
STRUCT
    UtcOffsetMin : DINT;   // local = UTC + offset. Set it; daylight saving is not guessed.
    StartMin     : ARRAY[1..PL_Fraktal.MAX_SHIFTS] OF DINT := [PL_Fraktal.MAX_SHIFTS(-1)];
                           // minutes after local midnight, -1 = shift not used
END_STRUCT
END_TYPE

// ---- DUTs/ST_ShiftRecord.TcDUT
// Core §8.5.2(b) - one closed shift, exactly as its figures stood at the boundary.
TYPE ST_ShiftRecord :
STRUCT
    ShiftIndex       : INT;     // 1..MAX_SHIFTS
    StartAt          : DT;      // §2.7 clock (UTC)
    EndAt            : DT;
    TimeSynchronized : BOOL;    // FALSE if either boundary was crossed on an unsynchronized clock
    ManualReset      : BOOL;    // counts or OEE were reset by hand during this shift
    GoodCount        : UDINT;
    NokCount         : UDINT;
    ReworkCount      : UDINT;
    RunMs            : UDINT;
    DownMs           : UDINT;
    IdleMs           : UDINT;
    Availability     : REAL;    AvailValid : BOOL;
    Performance      : REAL;    PerfValid  : BOOL;
    Quality          : REAL;    QualValid  : BOOL;
    Oee              : REAL;    OeeValid   : BOOL;
END_STRUCT
END_TYPE

// ---- DUTs/ST_LineRecord.TcDUT
// Core §3.8e - one line value as it travels from owner to mirror: the same
// (WriteKey, Revision, value text) a WRITE_CONFIG carries, so a mirror applies it
// through the ordinary typed handler and a revision mismatch refuses it.
TYPE ST_LineRecord :
STRUCT
    WriteKey  : STRING(160);
    Revision  : UDINT;
    ValueText : STRING(80);
END_STRUCT
END_TYPE

// ---- DUTs/ST_LineImage.TcDUT
// Core §3.8e - the owner's published line data, whole. A mirror reads this one
// structure and applies it all or not at all; nothing is ever read field by field.
TYPE ST_LineImage :
STRUCT
    LineId   : STRING(40);
    Owner    : STRING(80);   // owner module's canonical identity
    Revision : UDINT;        // rises on every accepted change at the owner
    Count    : INT;
    Records  : ARRAY[1..PL_Fraktal.MAX_LINE_RECORDS] OF ST_LineRecord;
END_STRUCT
END_TYPE

// ---- DUTs/ST_LineStatus.TcDUT
// Core §3.8e(d) - what a copy of line data says about itself.
TYPE ST_LineStatus :
STRUCT
    LineId      : STRING(40);
    Role        : E_LineRole;
    Owner       : STRING(80);   // identity of the copy this one came from
    Revision    : UDINT;        // revision held here
    LastUpdate  : DT;           // mirror: last successful update (§2.7 clock)
    TimeSynchronized : BOOL;    // quality of LastUpdate
    Stale       : BOOL;         // mirror: no successful update within the declared window
    SourceError : DINT;         // 0 ok; 1 wrong line; 2 not applicable whole; else source error
END_STRUCT
END_TYPE

// ---- DUTs/ST_ConfigAccess.TcDUT
// Core §3.8d - what a module declared about who may see and change
// one of its registered values. The ROOT turns this into an effective level
// with its policy; the module never decides policy, it only states the class
// and its own raise-only minimums.
TYPE ST_ConfigAccess :
STRUCT
    Kind          : E_ConfigKind;
    ClassId       : STRING(40);    // '' = the built-in class (DATA_READ/DATA_WRITE)
    MinReadLevel  : E_AccessLevel; // raise-only: never lowers the class level
    MinWriteLevel : E_AccessLevel;
END_STRUCT
END_TYPE

// ---- DUTs/ST_DataClassPolicy.TcDUT
// Core §3.8d - one project-declared data class: the ACCESS axis of
// editable data, orthogonal to its ConfigKind. The levels are policy (§7.7(b)):
// declared as defaults, persisted, and editable through ACCESS_POLICY.
TYPE ST_DataClassPolicy :
STRUCT
    ClassId    : STRING(40);    // stable identity a value is registered into
    LabelKey   : STRING(160);   // localization key for the class's name
    ReadLevel  : E_AccessLevel; // to see the class's values
    WriteLevel : E_AccessLevel; // to change them
END_STRUCT
END_TYPE

// ---- DUTs/ST_ConfigWriteDef.TcDUT
// Core §3.8b/§3.10.2 — one editable value a module has registered about itself.
// The module declares it once at Setup; the framework then both PUBLISHES the
// capability (M_AppendConfig) and APPLIES writes to it (M_ApplyConfigWrite) from
// this single record, so the metadata a client validates against and the target
// the PLC writes can never drift apart (§1.1 O1/O9).
//
// pTarget is a pointer held in ordinary VAR — never inside a persistent
// declaration, where TwinCAT would retain an address that means nothing after a
// restart (TC3 §3.8b).
TYPE ST_ConfigWriteDef :
STRUCT
    Key           : STRING(160);  // §3.10.2 WriteKey — the mutation identity
    Item          : STRING(255);  // browse/display fragment; never the write identity
    Revision      : UDINT;        // non-zero; bump when the value's meaning changes
    Kind          : E_ConfigKind;
    ValueType     : E_ConfigValueType;
    Storage       : E_ConfigStorage;
    pTarget       : PVOID;
    RequiresReady : BOOL;         // write refused unless the owning root is READY
    HasMinimum    : BOOL;
    HasMaximum    : BOOL;
    Minimum       : LREAL;
    Maximum       : LREAL;
    Unit          : E_EngUnit;    // a code; the HMI owns the symbol (std.unit.*)
    LabelKey      : STRING(160);
    MaxLength     : UINT;         // AS_STRING only: the target's declared capacity
    EnumDomain    : STRING(255);  // pipe-separated exact accepted values ('' = none)
    EnumLabelKey  : STRING(80);   // catalog prefix: value v is labelled '<key>.<v>'
    // §3.8c teach capture. The live source lives on the SAME record as the value
    // it writes, so a capture cannot reach a field that is not independently
    // editable - the back door §3.8c(a) forbids is structurally impossible here
    // rather than prevented by a check somebody could forget.
    // 0 = this value offers no capture, which is the default and most values.
    pCapture       : PVOID;
    CaptureStorage : E_ConfigStorage;   // how to READ the source (may differ from Storage)
    // §3.8d - the access axis. '' + NONE/NONE is the built-in class, which is
    // exactly the behaviour before data classes existed.
    ClassId       : STRING(40);
    MinReadLevel  : E_AccessLevel;
    MinWriteLevel : E_AccessLevel;
END_STRUCT
END_TYPE

// ---- DUTs/ST_ConfigEntry.TcDUT
// Core §3.10.2 — one configuration value served through the request mailbox
// instead of the cyclic OPC UA tree. Scope selects the owner ('' = the root
// Unit itself, a qualified dotted module identity for a child, '#Fieldbus' for
// the bus topology). Item is the value's browse fragment in the server's array
// naming (e.g. 'Catalog/Catalog[2]/Label') so a generic HMI can rebuild the
// exact published path it would otherwise have read. The append-only capability
// tail is fail-closed: Writable alone is insufficient; a client also requires a
// stable WriteKey and non-zero WriteRevision and the owning handler rechecks it.
TYPE ST_ConfigEntry :
STRUCT
    Scope     : STRING(255);
    Item      : STRING(255);
    ValueText : STRING(255);   // typed by the HMI from the Item vocabulary
    WriteKey      : STRING(160);
    WriteRevision : UDINT;
    ConfigKind    : E_ConfigKind;
    ValueType     : E_ConfigValueType;
    Writable      : BOOL;
    RequiresReady : BOOL;
    HasMinimum    : BOOL;
    HasMaximum    : BOOL;
    Minimum       : LREAL;
    Maximum       : LREAL;
    Unit          : STRING(16);
    LabelKey      : STRING(160);
    EnumDomain    : STRING(255); // pipe-separated exact accepted values
    // §3.8d - computed by the PLC so a client greys and hides from data, never
    // from its own copy of the policy. Readable = FALSE serves the entry WITHOUT
    // its value: the editor can say something exists and why it is hidden.
    ClassId       : STRING(40);
    ReadLevel     : E_AccessLevel;
    WriteLevel    : E_AccessLevel;
    Readable      : BOOL;
    // Appended (Core 0.14): the unit as a CODE the HMI translates, and the
    // catalog prefix that labels each EnumDomain value ('<key>.<value>'). Unit
    // above stays, derived from UnitCode, for clients that predate it.
    UnitCode      : E_EngUnit;
    EnumLabelKey  : STRING(80);
    // Appended (Core 0.19): TRUE for a model-data value in the root's own recipe
    // record. It follows the model a QUERY_CONFIG / WRITE_CONFIG names by index
    // (HmiRequest.DurationMs: 0 = the active model, n = AvailableModels[n]).
    ModelScoped   : BOOL;
END_STRUCT
END_TYPE

// ---- DUTs/ST_HmiResponse.TcDUT
// Core §3.10/§14 — acknowledgement for ST_HmiRequest.
TYPE ST_HmiResponse :
STRUCT
    AckSequence : UDINT;
    Accepted    : BOOL;           // request acted or query completed
    Diagnostic  : STRING(255);    // localization key when refused/unsupported
    Report      : ST_ReleaseReport;
    ConfigPage  : ST_ConfigPage;  // §3.10.2 QUERY_CONFIG page window
END_STRUCT
END_TYPE

// ---- DUTs/ST_HostEvent.TcDUT
// Core §11.6.2 — transport-neutral fixed host-event record. Optional strings are
// empty when not applicable; Sequence gives a north-bound adapter stable ordering.
TYPE ST_HostEvent :
STRUCT
    Sequence         : UDINT;
    Kind             : E_HostEventKind;
    StationPath      : STRING(255);
    PartUid          : STRING(64);
    Subject          : STRING(80);   // tool/resource/material identifier
    Value            : STRING(80);   // new mode/model/tool/material value
    Stamp            : DT;
    TimeSynchronized : BOOL;
    Verdict          : E_Verdict;
    ReasonCode       : E_Reason;
END_STRUCT
END_TYPE

// ---- DUTs/ST_IoChannel.TcDUT
// Core §10.5.1 — one fieldbus I/O channel (published for the topology view §3.13)
TYPE ST_IoChannel :
STRUCT
    // §3.10.2 — tag/wiring identity is activation-static: excluded from the
    // cyclic OPC UA tree and served via the config manifest. Live I/O state
    // (values, force, quality, fault) stays cyclically published.
    {attribute 'OPC.UA.DA' := '0'}
    Name       : STRING(80);
    {attribute 'OPC.UA.DA' := '0'}
    DescriptionKey : STRING(160); // project/standard localization key
    {attribute 'OPC.UA.DA' := '0'}
    Address    : STRING(80);    // physical locator, e.g. EL1809 Ch5
    {attribute 'OPC.UA.DA' := '0'}
    Path       : STRING(255);   // unique channel path (force/audit identity)
    {attribute 'OPC.UA.DA' := '0'}
    ModulePath : STRING(255);   // owning module browse path for cross-navigation
    {attribute 'OPC.UA.DA' := '0'}
    Dir        : E_ChannelDir;
    {attribute 'OPC.UA.DA' := '0'}
    Kind       : E_ChannelKind;
    BoolValue  : BOOL;          // digital
    AnalogValue: REAL;          // analog (scaled)
    {attribute 'OPC.UA.DA' := '0'}
    Unit       : STRING(16);
    Forced     : BOOL;
    Quality    : BOOL;          // TRUE = good
    FaultActive: BOOL;          // a module diagnostic implicates this exact channel
    Diagnostic : STRING(255);   // localization key; Name remains the exact I/O tag
    // Additive capability flag (Core 0.1.0.7). FALSE is the fail-closed default:
    // output direction alone never authorizes a raw process-image force. It is
    // also FALSE on every channel unless the §7.5 OUTPUT_FORCING gate is active,
    // which is what makes the HMI force affordance absent - not greyed - in a
    // production image (§3.9, §10.5.1 rule 1).
    {attribute 'OPC.UA.DA' := '0'}
    Forceable  : BOOL;
    // §10.5.1 - the HELD force set-point. Kept apart from BoolValue/AnalogValue
    // on purpose: those are overwritten every scan by the hardware driver's
    // publish, so a set-point stored there would survive exactly one cycle, and
    // clearing a force would freeze the last forced value instead of restoring
    // the real one. Commissioning data, never cyclically published.
    {attribute 'OPC.UA.DA' := '0'}
    ForceBool  : BOOL;
    {attribute 'OPC.UA.DA' := '0'}
    ForceAnalog: REAL;
END_STRUCT
END_TYPE

// ---- DUTs/ST_ModuleStatus.TcDUT
// Core §3.10(a')/§3.12/§6.9(a) — the DATA MIRROR every module publishes each scan.
// Properties/methods serve PLC code; this struct serves OPC UA/HMI. It is the
// framework baseline of the OutImm role: name, tier, state summary, and the live
// first-out diagnostic — everything a generic tile needs, browsable by type.
TYPE ST_ModuleStatus :
STRUCT
    Name        : STRING(80);     // = browse name (§4.8) — the tile caption
    DisplayNameKey : STRING(160); // optional localization key; Name remains identity
    DescriptionKey : STRING(160); // optional module information localization key
    TypeKey     : STRING(160);    // §7.1 type key: one per TYPE, not per instance; '' = coarse ModuleType scope
    ModuleType  : E_ModuleType;   // UNIT | EQUIPMENT_MODULE | CONTROL_MODULE (tile kind)
    State       : E_ExecState;    // the tile state LED
    FaultActive : BOOL;
    Diagnostic  : ST_Diagnostic;  // live first-out (§6.9(a)) — the tile message line
    TileEnable  : BOOL := TRUE;   // §3.13: render as a tile on the parent's child view
    ControlDomainId : STRING(80); // §9.8: '' = no safety/control-power arrangement
END_STRUCT
END_TYPE

// ---- DUTs/ST_PartResult.TcDUT
// Core §3.16.1
TYPE ST_PartResult :
STRUCT
    Verdict     : E_Verdict;     // NONE | OK | NOK | REWORK
    ReasonCode  : E_Reason;      // first NOK reason — SAME vocabulary as a fault (Core §8.8)
    Records     : ARRAY[1..PL_Fraktal.MAX_RESULTS] OF ST_MeasRecord;
    StationPath : STRING(255);   // browse path of the producing station (Core §4.8)
    Stamp       : DT;            // synchronized timestamp (Core §2.7)
    TimeSynchronized : BOOL;
END_STRUCT
END_TYPE

// ---- DUTs/ST_StepRecord.TcDUT
// Core §6.5 — what the stall walk reads
TYPE ST_StepRecord :
STRUCT
    StepNo        : INT;
    StepName      : STRING(120);   // localization key
    AwaitingLabel : STRING(120);   // e.g. 'ClampStation.CLAMP' ('' if none)
    TimeClass     : E_TimeClass;   // Core §8.11.4(f) — WORK unless a genuine wait
    ExpectedTime  : TIME;          // defaults from the awaited command's timeout
    Conds         : ARRAY[1..PL_Fraktal.MAX_STEP_CONDS] OF ST_CondRecord;
END_STRUCT
END_TYPE

// ---- DUTs/ST_StateFlag.TcDUT
// Core §3.12 — one published DERIVED state flag.
//
// The distinction it enforces: `OutCmd` is what a command PRODUCED, latched
// until the next command; a state flag is what is TRUE RIGHT NOW, recomputed
// from the modules underneath every scan. `Homed` is the worked example - as a
// command result it keeps claiming "homed" after an operator jogs an axis off
// home in MANUAL, because no sequence runs to clear the latch. As a derived flag
// it simply stops being true.
TYPE ST_StateFlag :
STRUCT
    Key   : STRING(120);   // localization key; '' = slot never published
    Value : BOOL;
    // When Value last changed, on the synchronized clock (§2.7). This is what a
    // bare assignment cannot give and the operator always asks for: not just
    // "is the door closed" but "how long has it been closed".
    Since : DT;
    // The owner stopped publishing this flag - it was computed behind an IF that
    // stopped being true, or the code that produced it was removed. Value is
    // forced FALSE: a flag nobody is computing is not a claim (§5.6 fail-safe).
    Stale : BOOL;
END_STRUCT
END_TYPE

// ---- DUTs/ST_SequenceStepDef.TcDUT
// Core §3.13/§3.10.2 — the STATIC definition of a flow-chart row.
//
// Every field here is fixed from the step's first visit, so none of it belongs in a
// cyclic read. It is served through the config manifest (M_AppendConfig) under the
// SAME browse paths the live row uses, so the HMI reads one row structure and never
// learns that half of it arrived once and was cached.
TYPE ST_SequenceStepDef :
STRUCT
    StepNo        : INT;
    // §6.12 which concurrent leg this step belongs to. 0 = the chain's main line.
    Branch        : INT;
    TimeClass     : E_TimeClass;
    ExpectedTime  : TIME;          // 0 = no declared guard
    StepName      : STRING(120);   // localization key
    AwaitingLabel : STRING(120);   // e.g. 'PressRam.EXTEND' ('' if none)
    // §3.13 drill-down target: the Fraktal path of the module this step commands.
    // STRING(80) because that is what it is copied from - I_Module.Name, backed by
    // FB_ModuleBase._name : STRING(80). A module path cannot be longer than its own
    // name, so 255 was reserving 175 bytes per row that could never be used.
    AwaitsPath    : STRING(80);
END_STRUCT
END_TYPE

// ---- DUTs/ST_SequenceCursor.TcDUT
// Core §3.13/§6.12 — which row a concurrent leg is running, and for how long.
//
// Indexed BY BRANCH, because a leg has exactly one active step by definition: index
// 0 is the chain's main line, 1..n are its parallel legs. That is what makes this
// table ~10 entries instead of one per row, and small enough to publish cyclically -
// so the chart is already correct the instant its tab opens, instead of after the
// first on-demand read.
TYPE ST_SequenceCursor :
STRUCT
    RowIdx   : INT;                // SequenceSteps index; 0 = this leg has no active step
    Elapsed  : TIME;               // how long that row has been running
    TimedOut : BOOL;               // it outran its own ExpectedTime (a leg's own guard)
END_STRUCT
END_TYPE

// ---- DUTs/ST_SequenceAnnotation.TcDUT
// Core §6.9 — one error or message currently attached to a flow-chart row.
//
// These are SPARSE: an error is one at a time, and messages last only until their
// step is entered again, so a handful are live at once out of a table of 128 rows.
// Reserving the text on every row cost 633 of the row's 1156 bytes for a case that
// is almost always empty. The row keeps the flag; this carries what it says.
TYPE ST_SequenceAnnotation :
STRUCT
    RowIdx     : INT;              // SequenceSteps index this belongs to; 0 = free slot
    IsError    : BOOL;             // TRUE = §6.9(d) raise (chain stopped), FALSE = §6.9(e) message
    Key        : STRING(120);      // localization key of the reason/message
    // Module the chart drills into; '' = this Unit. STRING(80) for the same reason
    // as AwaitsPath: it is a module path, bounded by FB_ModuleBase._name.
    SourcePath : STRING(80);
END_STRUCT
END_TYPE

// ---- DUTs/ST_SequenceStep.TcDUT
// Core §6.5/§3.13 — the per-row LIVE state of one flow-chart row: 7 bytes.
//
// Everything static about a row (its number, leg, time class, guard and text) is in
// ST_SequenceStepDef, served once through the §3.10.2 manifest. Everything about
// which row is running RIGHT NOW is in ST_SequenceCursor, one entry per concurrent
// leg. What is left here is the small set that is per-row AND changes over time,
// and that the HMI could not reconstruct by watching: a poll at a few Hz against a
// task at kHz cannot see a step shorter than its own interval, so a chart that
// accumulated these client-side would silently skip fast steps and lose transient
// errors. The chart shows what the chain DID, not what someone happened to catch.
TYPE ST_SequenceStep :
STRUCT
    Visited       : BOOL;          // reached at least once since the chain reset
    LastDuration  : TIME;          // how long it ran on its last visit
    // §6.9(d)/(e) marks. The text and the drill-down link are in the annotation
    // table; these say only that the row has one, which is all the chart needs to
    // colour it - so a row stays correctly marked even if that table is full.
    ErrorActive   : BOOL;
    WarningActive : BOOL;
END_STRUCT
END_TYPE

// ---- DUTs/ST_StepTiming.TcDUT
// Core §8.11.4(b)/(f) — one step of a cycle profile (Gantt/waterfall row)
TYPE ST_StepTiming :
STRUCT
    StepNo   : INT;
    StepName : STRING(120);   // localization key
    TimeClass    : E_TimeClass;  // WORK unless the step declared a wait class (§8.11.4(f))
    Started  : DT;           // synchronized wall clock (Core §2.7) — aligns across stations
    StartedTimeSynchronized : BOOL;
    Duration : TIME;         // monotonic-clock duration (TC3 §8.11)
    Expected : TIME;         // §8.11.4(c) — the step's declared guard, drawn vs actual (0 = none)
END_STRUCT
END_TYPE

// ---- DUTs/ST_SignalTowerOut.TcDUT
// Core §8.13 — semantic HAL output; a project Hardware Driver owns channel maps.
TYPE ST_SignalTowerOut :
STRUCT
    Red      : BOOL;
    Amber    : BOOL;
    Green    : BOOL;
    Blue     : BOOL;
    White    : BOOL;
    Horn     : BOOL;
    TestActive : BOOL;
END_STRUCT
END_TYPE

// ---- DUTs/ST_SignalTowerParCfg.TcDUT
// Core §8.13 — the site convention changes configuration, not mapping code.
TYPE ST_SignalTowerParCfg :
STRUCT
    SchemaVersion     : UINT := 1;
    LampTestDuration  : TIME := T#3S;
    OperatorUsesWhite : BOOL;
    HornOnHigh        : BOOL := TRUE;
END_STRUCT
END_TYPE

// ---- DUTs/ST_SystemHealthInput.TcDUT
// Core §8.12 — platform-neutral probe sample. Availability is explicit so an
// unsupported metric never masquerades as a healthy zero.
TYPE ST_SystemHealthInput :
STRUCT
    TaskAvailable       : BOOL;
    TaskCycleUs         : UDINT;
    TaskJitterUs        : UDINT;
    TaskOverrun         : BOOL;
    ControllerAvailable : BOOL;
    CpuLoadPct          : LREAL;
    MemoryAvailableMb   : UDINT;
    IpcAvailable        : BOOL;
    IpcTemperatureC     : LREAL;
    FanHealthy          : BOOL;
    StorageHealthPct    : LREAL;
    FieldbusAvailable   : BOOL;
    FieldbusMasterHealthy : BOOL;
    LostFrameCount      : UDINT;
    SlaveErrorCount     : UDINT;
    DcAvailable         : BOOL;
    DcSynchronized      : BOOL;
    TimeQuality         : ST_TimeQuality;
    // Per-metric availability inside the IPC group (Core §8.12: "where the hardware
    // exposes them"). TRUE by default, so a producer that sets only IpcAvailable
    // keeps its meaning; a target provider clears the one it cannot measure - a
    // fanless IPC, a drive without flash wear data - instead of inventing a value.
    FanAvailable        : BOOL := TRUE;
    StorageAvailable    : BOOL := TRUE;
END_STRUCT
END_TYPE

// ---- DUTs/ST_SystemHealthParCfg.TcDUT
// Core §8.12 — station-selected health thresholds. SchemaVersion is first
// because this record follows the same migrate-or-fault rule as every ParCfg.
TYPE ST_SystemHealthParCfg :
STRUCT
    SchemaVersion        : UINT := 1;
    MaxTaskCycleUs       : UDINT := 100000;
    MaxTaskJitterUs      : UDINT := 10000;
    MaxCpuLoadPct        : LREAL := 90.0;
    MinMemoryAvailableMb : UDINT := 128;
    MaxIpcTemperatureC   : LREAL := 80.0;
    MinStorageHealthPct  : LREAL := 10.0;
    MaxLostFrames        : UDINT := 0;
    MaxSlaveErrors       : UDINT := 0;
    MaxTimeOffsetUs      : DINT := 1000;
    RequireFieldbus      : BOOL;
    RequireDcSync        : BOOL;
    RequireTimeSync      : BOOL := TRUE;
END_STRUCT
END_TYPE

// ---- DUTs/ST_SystemHealthStatus.TcDUT
// Core §8.12 — small cyclic health surface for OPC UA trending. Raw probes are
// hidden; this validated copy is the public contract.
TYPE ST_SystemHealthStatus :
STRUCT
    Present             : BOOL;
    Healthy             : BOOL;
    SourcePath          : STRING(255);
    TaskAvailable       : BOOL;
    TaskCycleUs         : UDINT;
    TaskJitterUs        : UDINT;
    TaskOverrun         : BOOL;
    ControllerAvailable : BOOL;
    CpuLoadPct          : LREAL;
    MemoryAvailableMb   : UDINT;
    IpcAvailable        : BOOL;
    IpcTemperatureC     : LREAL;
    FanHealthy          : BOOL;
    StorageHealthPct    : LREAL;
    FieldbusAvailable   : BOOL;
    FieldbusMasterHealthy : BOOL;
    LostFrameCount      : UDINT;
    SlaveErrorCount     : UDINT;
    DcAvailable         : BOOL;
    DcSynchronized      : BOOL;
    TimeQuality         : ST_TimeQuality;
    FanAvailable        : BOOL;     // FanHealthy is a measurement
    StorageAvailable    : BOOL;     // StorageHealthPct is a measurement
END_STRUCT
END_TYPE

// ---- DUTs/ST_TimeQuality.TcDUT
// Core §2.7 — quality of the one PLC wall clock used by every Fraktal stamp.
// Available=FALSE is deliberately not equivalent to synchronized.
TYPE ST_TimeQuality :
STRUCT
    Available    : BOOL;
    Synchronized : BOOL;
    Source       : STRING(32);   // documented station source: PTP, DC, NTP, ...
    OffsetUs     : DINT;         // signed offset from the selected source
    LastSyncAt   : DT;
    ObservedAt   : DT;
END_STRUCT
END_TYPE

// ---- DUTs/ST_TimingRow.TcDUT
// Core §8.11.4 — one timing aggregate, keyed by command id (a) or StepNo (b)
TYPE ST_TimingRow :
STRUCT
    Id        : DINT;         // TO_DINT(E_<Type>Command) or StepNo; 0 = untagged
    Label     : STRING(120);   // command/step localization key for the HMI table
    TimeClass : E_TimeClass;  // §8.11.4(f); commands are WORK by definition
    Count     : UDINT;        // completed executions (0 = row unused)
    Last      : TIME;
    Minimum   : TIME;
    Maximum   : TIME;
    Avg       : TIME;         // running mean (F_TimingUpdate)
END_STRUCT
END_TYPE

// ---- DUTs/ST_UserRecord.TcDUT
// Core §7.7(c) — FB_LocalAccessProvider table entry (local default; server-side
// auth substitutes via I_AccessProvider without touching module code). Packed:
// it is also the record of the retained ST_AccessImageV1.
{attribute 'pack_mode' := '1'}
TYPE ST_UserRecord :
STRUCT
    User    : STRING(32);
    // §14 - the PIN itself is never stored: a salt drawn at registration and the
    // iterated SHA-256 of salt and PIN (FB_LocalAccessProvider._M_Hash).
    Salt    : ARRAY[0..15] OF BYTE;
    PinHash : ARRAY[0..31] OF BYTE;
    Level   : E_AccessLevel;
END_STRUCT
END_TYPE

// ---- DUTs/ST_AccessImageV1.TcDUT
// Core §7.7(c)/§14 - FB_LocalAccessProvider's retained user table as it is kept
// in the TwinCAT Boot directory: fixed-width, packed (identical on x86/x64/Arm),
// versioned and CRC-protected, so a torn, foreign or edited file is rejected as a
// whole instead of being half-restored. It carries salts and PIN hashes only.
{attribute 'pack_mode' := '1'}
TYPE ST_AccessImageV1 :
STRUCT
    SchemaVersion : UINT;      // 1
    ByteCount     : UINT;      // SIZEOF(ST_AccessImageV1)
    Magic         : DWORD;     // 'FRKA'
    Generation    : UDINT;     // increases with every durable write
    Count         : INT;       // valid entries in Users
    Reserved      : INT;       // 0
    Users         : ARRAY[1..PL_Fraktal.MAX_USERS] OF ST_UserRecord;
    Crc           : DWORD;     // F_Crc32 of every byte before this field
END_STRUCT
END_TYPE

// ---- DUTs/ST_PersistResult.TcDUT
// Core §3.8b - the outcome of one I_PersistMedium request.
TYPE ST_PersistResult :
STRUCT
    Ok      : BOOL;    // write: durable. read: the medium answered (Found or not)
    Found   : BOOL;    // read: a valid, non-empty document was returned
    Lost    : BOOL;    // read: a document this medium confirmed writing is missing,
                       // corrupt or older than confirmed - something was lost
    Length  : UDINT;   // read: bytes returned
    ErrorId : UDINT;   // last medium error (0 = none)
END_STRUCT
END_TYPE

// ---- DUTs/ST_RetainDocument.TcDUT
// Core §3.8b - one document in FB_RetainPersistMedium's persistent pool.
TYPE ST_RetainDocument :
STRUCT
    Key        : STRING(80);     // '' = free slot
    Generation : UDINT;          // increases with every write of this key
    Length     : UDINT;
    Crc        : DWORD;          // F_Crc32 of Data[0..Length-1]
    Data       : ARRAY[0..PL_Fraktal.MAX_PERSIST_DOC_BYTES - 1] OF BYTE;
END_STRUCT
END_TYPE

// ---- DUTs/ST_TcpVisionOutImm.TcDUT
TYPE ST_TcpVisionOutImm :
STRUCT
    LinkState    : E_ByteChannelState;
    LastResponse : STRING(255);
END_STRUCT
END_TYPE

// ---- DUTs/ST_TcpCodeReaderOutImm.TcDUT
TYPE ST_TcpCodeReaderOutImm :
STRUCT
    LinkState    : E_ByteChannelState;
    LastResponse : STRING(255);
END_STRUCT
END_TYPE

// ---- DUTs/ST_TcWindowsClockSampleV1.TcDUT
// Fixed-width Windows observer wire record: 76 bytes on x86/x64.
{attribute 'pack_mode' := '1'}
TYPE ST_TcWindowsClockSampleV1 :
STRUCT
    SchemaVersion  : UINT;
    ByteCount      : UINT;
    Magic          : DWORD;
    Sequence       : UDINT;
    ObservedAt     : DT;
    LastSyncAt     : DT;
    OffsetUs       : DINT;
    SyncAgeSeconds : UDINT;
    ServiceError   : UDINT;
    Flags          : DWORD;
    Source         : STRING(32);
    ReservedBytes  : ARRAY[0..2] OF BYTE;
    Crc            : DWORD;
END_STRUCT
END_TYPE

// ---- Params/PL_Fraktal.TcGVL
{attribute 'qualified_only'}
// Fraktal Core — framework constants (Core §7.2, §3.2, §6.5, §3.16, §6.11)
VAR_GLOBAL CONSTANT
    MAX_PERMINTLK_COND   : INT := 16;   // Core §7.2 (default 16)
    MAX_EM_CHILDREN      : INT := 16;
    MAX_SEQUENCES        : INT := 16;
    // Core §3.13 — rows in a published sequence flow chart. 32 covered the demo but
    // not a real machine: a station chain of a hundred-odd steps is ordinary, and the
    // overflow is SILENT (the row is dropped, the chart just stops growing).
    //
    // The cost is per Unit and it is nearly all strings: one row is ~1.16 kB, of which
    // 98% is the five localization-key and path fields. 128 rows is ~145 kB of PLC
    // memory per Unit and 2176 OPC UA nodes, which is why SequenceSteps is an
    // ON-DEMAND subtree on the HMI side (read while the Sequence tab is open, never in
    // the cyclic snapshot) - see Specification/HMI_CONTRACT.md. Raising this further
    // costs linearly in both; shortening the string fields is the lever if it matters.
    MAX_SEQUENCE_STEPS   : INT := 128;
    // Core §6.9 — errors/messages attached to flow-chart rows at once. Sparse by
    // nature (one error; a message per step visit until that step runs again), so
    // this is far below MAX_SEQUENCE_STEPS on purpose. If it fills, the row keeps
    // its mark and loses only the text (§5.6 degrade, never mislead).
    MAX_SEQUENCE_ANNOTATIONS : INT := 16;   // Core §6.8 — chains attached to one Unit (incl. sub-chains)   // Core §3.2 / §8.2
    MAX_STEP_CONDS       : INT := 8;    // Core §6.9(b) condition records per step
    // Core §3.12 — derived state flags a module may publish. Statically sized
    // per module like every other Fraktal table (§1.1 O10).
    MAX_STATE_FLAGS      : INT := 12;
    MAX_GENEALOGY        : INT := 8;    // Core §3.16.1
    MAX_RESULTS          : INT := 32;   // Core §3.16.1
    MAX_OPTIONS          : INT := 6;    // Core §6.11
    MAX_CMD_STATS        : INT := 8;    // Core §8.11.4(a) — distinct command ids per module
    MAX_PROFILE_STEPS    : INT := 32;   // Core §8.11.4(b) — steps per cycle profile
    MAX_RECIPES          : INT := 16;   // Core §3.8 — records per FB_LocalRecipeProvider
    MAX_MODEL_DATA_BYTES : UDINT := 1024; // Core §3.8a — a Unit's own recipe record, edited per model
    MAX_MODEL_FIELDS     : INT := 8;    // Core §3.8a — client-defined named model fields
    MAX_ALARM_ACTIVE     : INT := 16;   // Core §8.3 — concurrently open events per Unit
    MAX_ALARM_RING       : INT := 64;   // Core §8.3 — closed-event history ring per Unit
    MAX_HOST_EVENTS      : INT := 32;   // Core §11.6 — per-Unit north-bound event ring
    MAX_USERS            : INT := 16;   // Core §7.7 — FB_LocalAccessProvider user table
    PIN_HASH_ROUNDS      : UINT := 256; // §14 — extra SHA-256 rounds per stored PIN (one login ~1 ms)
    MAX_POS_SENSORS      : INT := 2;    // redundant sensors per cylinder position (duplex; raise for 2oo3)
    MAX_NODE_CHANNELS    : INT := 16;   // Core §10.5.1 — I/O channels per fieldbus node
    MAX_BUS_NODES        : INT := 64;   // Core §10.5.1 — nodes in the flat topology table
    // Core §7.5.1 — commissioning/engineering gates one station may declare.
    // Small on purpose: a station carrying more than a handful of deliberate
    // departures from its production configuration has a process problem, not a
    // table-size problem. Overflow sets FB_EngineeringMode.Truncated (§5.6).
    MAX_ENGINEERING_GATES : INT := 8;
    MAX_CMD_CATALOG      : INT := 12;   // Core §7.6.1 — manual commands a module may publish
    MODE_COUNT           : INT := 7;    // Core §3.4 — E_Mode entries (AUTO..ADJUSTMENT), for policy array
    MAX_RELEASE_REASONS  : INT := 24;   // Core §7.8 — entries in a release report
    MAX_OEE_SAMPLES      : INT := 60;      // Core §8.5.1 — trend ring length
    MAX_CYCLE_HISTORY    : INT := 60;      // Core §8.11.4 — per-cycle summary ring (trend charts)
    OEE_SAMPLE_MS        : UDINT := 60000; // Core §8.5.1 — sample period (1 min)
    MAX_ALARM_META       : INT := 32;      // Core §8.9 — rationalization records per log
    MAX_SHELF_S          : UDINT := 28800; // Core §8.10 — shelf cap (8h)
    MAX_DIAG_RING        : INT := 16;   // Core §6.9(a) — Unit diagnostic history depth
    MAX_CONFIG_PAGE      : INT := 16;   // Core §3.10.2 — config-manifest entries per mailbox page
    MAX_CONFIG_WRITES    : INT := 12;   // Core §3.8b — editable values one module may register
    // Core §3.8b — named parameter sets held by FB_LocalConfigStore, and records
    // per set. Both cost PERSISTENT memory directly: one record is ~340 B, so the
    // shipped 4 × 32 reserves roughly 44 kB of the controller's persistent budget.
    // A deployment needing more sizes the PLC persistent area to match, or wires a
    // FILE_JSON/EXTERNAL store instead — the framework never grows this at run time.
    MAX_CONFIG_SETS      : INT := 4;
    MAX_DATA_CLASSES     : INT := 8;
    MAX_LINE_RECORDS     : INT := 32;
    MAX_WEEKLY_SHIFTS    : INT := 5; // additive V3 capacity; daily layout stays four
    MAX_SHIFTS           : INT := 4;   // §8.5.2 shifts in a line's calendar
    MAX_SHIFT_HISTORY    : INT := 8;   // §8.5.2 closed shifts a Unit keeps  // §3.8e values one line carries   // §3.8d project-declared data classes per root
    MAX_SET_RECORDS      : INT := 32;
    // Core §3.8b — the DECLARED bounded window an accepted configuration write has
    // to reach non-volatile storage. Publishing the number is the point: "durability
    // is a stated property, not a hope", and a station whose store cannot meet it
    // says so through PersistFailed instead of reverting silently at the next start.
    CONFIG_PERSIST_WINDOW_MS : UDINT := 5000;
    // Core §3.8b — one retained DOCUMENT on an I_PersistMedium: a rendered set (a
    // header and MAX_SET_RECORDS lines of at most 480 characters fit) or the user
    // table's image. Every FB_ConfigSetDocument holds one buffer of this size.
    MAX_PERSIST_DOC_BYTES : UDINT := 16384;
    MAX_PERSIST_QUEUE    : INT := 8;    // requests one medium holds at once (FIFO)
    MAX_PERSIST_KEYS     : INT := 48;   // documents a file medium vouches for (loss detection)
    MAX_RETAIN_DOCUMENTS : INT := 8;    // FB_RetainPersistMedium pool: 8 x 16 kB persistent
    // Core §7.6.1a — how long a latched hold-to-run request survives without a
    // refresh from the client. Long enough to ride out transport jitter, short
    // enough that a closed HMI or a dead link lets go rather than leaving the
    // machine moving. The module's own JogTimeout is the second, shorter net.
    MANUAL_HELD_REFRESH_MS : DWORD := 750;
    // Core §3.13/§3.10.2 — how long the flow chart must stop growing before the
    // manifest revision is raised for it.
    //
    // §3.13 rows are discovered by VISIT, one at a time, while the manifest is
    // invalidated ALL AT ONCE. A per-row bump therefore asked a client to
    // refetch the entire manifest once per row: entering AUTO on the press
    // discovers 15 rows where HOME discovers 2, which is why HOME->AUTO stalled
    // and HOME->HOME did not.
    //
    // Waiting for the burst to settle is strictly better than bumping per row,
    // on BOTH counts: far fewer refetches, and the client fetches AFTER the
    // chart stops growing rather than during it - which is the very failure the
    // per-row bump was written to avoid ("a chart that grows after the HMI's
    // fetch would render every new row with StepNo 0 and no text").
    CHART_REV_SETTLE_MS : DWORD := 1000;
    MAX_SAFETY_DEVICES   : INT := 16;   // Core §9 — published safety aliases per module/zone
    MAX_POWER_GROUPS     : INT := 8;    // Core §9 — independently controlled energy groups
    MAX_CONTROL_DOMAIN_UNITS : INT := 16; // Core §9.8 — root Units sharing one arrangement
    // Core §6.12 — concurrent legs one chain may run at once. It bounds the
    // per-leg transition results AND every per-leg step-scoped latch, so it is a
    // real memory cost per chain, not a loop limit (§1.1 O10: statically sized,
    // no run-time allocation). Legs are numbered 1..n; 0 is the main line and is
    // always available on top of these.
    MAX_PARALLEL_BRANCHES : INT := 9;
    // TC3 Windows observer default, also emitted into the observer package.
    WINDOWS_CLOCK_SAMPLE_FILE : STRING(255) := 'C:\ProgramData\Fraktal\Clock\quality.bin';
END_VAR

// ---- GVLs/GVL_FraktalTime.TcGVL
{attribute 'qualified_only'}
VAR_GLOBAL
    // One PLC-wide clock-quality authority. Hidden here; each root republishes
    // the validated value beside its system-health surface.
    {attribute 'OPC.UA.DA' := '0'}
    Current : ST_TimeQuality;
END_VAR

// ---- Params/PL_FraktalCompat.TcGVL
{attribute 'qualified_only'}
// Fraktal Core — TwinCAT compiler-compatibility policy (O8 portable, O9 one
// authoritative source, O1 low developer effort).
//
// ---------------------------------------------------------------------------
// POLICY
// ---------------------------------------------------------------------------
// The library targets MODERN TwinCAT (>= 3.1.4026) by default and treats
// 3.1.4024 as a supported LEGACY target. Modern language features are used
// freely; where a feature is unavailable on 4024, the legacy form is selected by
// a conditional pragma keyed on ONE compiler define:
//
//     FRAKTAL_TC3_4024
//
// Absent  (default) -> modern: defaulted METHOD inputs, etc.
// Defined           -> legacy 4024: the conservative form.
//
// This inverts the previous policy, where 4024 was the ceiling for everyone and
// every developer paid its restrictions (e.g. repeating `OnJump1 := -1,
// OnJump2 := -1, OnJump3 := -1` at all 22 M_Advance call sites).
//
// ---------------------------------------------------------------------------
// HOW TO BUILD FOR LEGACY 4024
// ---------------------------------------------------------------------------
// Add the define to EVERY PLC project in the solution (the library AND the
// application, since a pragma is evaluated per compiled project):
//
//   XAE: PLC project -> Properties -> Compile -> "Compiler Defines"
//        enter:  FRAKTAL_TC3_4024
//
//   or in the .plcproj PropertyGroup:
//        <CompilerDefines>FRAKTAL_TC3_4024</CompilerDefines>
//
// Verify with: python FraktalCore/PLC/TwinCAT/tools/plc_lint.py --profile 4024
// (that profile fails on any modern-only construct that is NOT pragma-guarded).
//
// ---------------------------------------------------------------------------
// FEATURES GUARDED TODAY
// ---------------------------------------------------------------------------
// 1. Defaulted METHOD VAR_INPUT  (requires >= 3.1.4026)
//    On 4024 a defaulted input still makes the argument MANDATORY at the call
//    site, so a caller that omits it fails with
//        "M_Advance requires exactly 'N' inputs"
//    Guarded in: FB_SequenceBase.M_Advance (OnJump1..3), .M_ResetBase (FirstStep)
//
// Conditional pragmas themselves are available in the DECLARATION part from
// 3.1.4024 onward, so the guard mechanism works on both targets.
// Reference: infosys.beckhoff.com "Conditional pragmas" (tc3_plc_intro).
//
// ---------------------------------------------------------------------------
// ADDING A NEW GUARDED FEATURE
// ---------------------------------------------------------------------------
//   {IF defined (FRAKTAL_TC3_4024)}
//   // legacy form
//   {ELSE}
//   // modern form
//   {END_IF}
//
// Rules: keep the MODERN form in the {ELSE} branch (it is the default target);
// make the legacy branch behaviour-identical, never merely compilable; and list
// the feature above so this file stays the single source of truth for the policy.
VAR_GLOBAL CONSTANT
    // Mirror of the build's compatibility mode, readable from code and visible on
    // the HMI/ADS surface so a deployed binary can be identified without
    // inspecting project settings.
    {IF defined (FRAKTAL_TC3_4024)}
    LEGACY_TC3_4024      : BOOL := TRUE;
    COMPAT_PROFILE       : STRING(16) := '4024-legacy';
    {ELSE}
    LEGACY_TC3_4024      : BOOL := FALSE;
    COMPAT_PROFILE       : STRING(16) := '4026-modern';
    {END_IF}
END_VAR

// ---- Params/PL_FraktalEngineering.TcGVL
{attribute 'qualified_only'}
// Fraktal Core — the framework's own commissioning/engineering build gates
// (Core §7.5.1, TC3 §7.5).
//
// ---------------------------------------------------------------------------
// WHY THESE ARE VAR_GLOBAL CONSTANT
// ---------------------------------------------------------------------------
// §7.5.1 requires a gate to be a BUILD constant, never a runtime variable:
// defeating one must be a source change plus a download — a reviewable, auditable
// act — and never an online write from an HMI, an ADS client or any other data
// path. The compiler also inlines a constant, so there is usually no symbol for a
// client to write at all. Do not "helpfully" convert these to writable variables,
// and do not add a writable mirror with a consumer in control logic.
//
// The application's own gates (USE_SIMULATION, CONTROL_CIRCUIT_MAPPING_CONFIRMED,
// …) stay where they are — in that project's MAIN — and are declared into the
// same register through FB_EngineeringMode.M_Declare. This GVL holds only the
// gates the FRAMEWORK owns.
//
// ---------------------------------------------------------------------------
// HOW TO BUILD A COMMISSIONING (ENGINEERING) IMAGE
// ---------------------------------------------------------------------------
// Add the define to EVERY PLC project in the solution — a conditional pragma is
// evaluated per compiled project, so the library and the application must agree:
//
//   XAE: PLC project -> Properties -> Compile -> "Compiler Defines"
//        enter:  FRAKTAL_ENGINEERING
//
//   or in the .plcproj PropertyGroup:
//        <CompilerDefines>FRAKTAL_ENGINEERING</CompilerDefines>
//
// A production image is simply one built WITHOUT that define. It is not a
// configuration a commissioning engineer can change on the machine.
VAR_GLOBAL CONSTANT
    // Core §10.5.1 rule 1 — may this image force fieldbus OUTPUT channels from
    // the HMI at all? FALSE keeps Forceable FALSE on every channel, so the HMI
    // renders no force affordance whatsoever (§3.9), and FB_UnitBase.ForceChannel
    // refuses every request before the resolver is ever reached.
    //
    // Forcing an INPUT is not offered by this surface in either build (§10.5.1
    // rule 2): lying to the logic to bypass a sensor or an interlock is an
    // engineering-tool act under separate authority, never an operating practice.
{IF defined (FRAKTAL_ENGINEERING)}
    OUTPUT_FORCING : BOOL := TRUE;
{ELSE}
    OUTPUT_FORCING : BOOL := FALSE;
{END_IF}
END_VAR

// ---- Params/PL_ReasonCatalog.TcGVL
{attribute 'qualified_only'}
// GENERATED FILE — DO NOT EDIT. §8.8/§8.9 catalog size.
VAR_GLOBAL CONSTANT
    COUNT : INT := 77;
END_VAR

// ---- Interfaces/I_RecipeCatalog.TcIO
// Optional bounded creation, discovered on I_RecipeProvider. The root validates
// the complete typed model projection before this provider commits storage.
INTERFACE I_RecipeCatalog

METHOD M_ModelCount : INT
VAR_INPUT
    RecipeKey : STRING(80);
END_VAR
END_METHOD

METHOD M_ModelCapacity : INT
VAR_INPUT
    RecipeKey : STRING(80);
END_VAR
END_METHOD

METHOD M_ModelAt : BOOL
VAR_INPUT
    RecipeKey : STRING(80);
    Index : INT;
END_VAR
VAR_IN_OUT
    Id : ST_ModelId;
END_VAR
END_METHOD

METHOD M_CreateModel : BOOL
VAR_INPUT
    ModelCode : STRING(64);
    RecipeKey : STRING(80);
    pData : PVOID;
    Size : UDINT;
END_VAR
END_METHOD

METHOD M_TakeCatalogRestoreLoss : BOOL
VAR_OUTPUT
    Found : UINT;
END_VAR
END_METHOD

END_INTERFACE

// ---- Interfaces/I_LineSource.TcIO
// Core §3.8e(c) - where a mirror gets its owner's line data from. Pluggable
// like §3.8's recipe provider and §3.8b's store; the transport is a binding and
// deployment choice, and what it returns is untrusted input (§14).
INTERFACE I_LineSource

// Call every scan. TRUE on the scan a complete owner image was obtained.
METHOD M_Poll : BOOL
VAR_IN_OUT
    Image : ST_LineImage;
END_VAR
END_METHOD

// The last transport error, 0 when the last attempt succeeded.
METHOD M_Error : DINT
END_METHOD

END_INTERFACE

// ---- Interfaces/I_AccessProvider.TcIO
// Core §7.7(c) — credential validation, injectable like every provider (§3.8).
// Returns the granted level; NONE = authentication failed. A provider may also
// implement I_AccessStore (a durable table), found by __QUERYINTERFACE.
INTERFACE I_AccessProvider EXTENDS __System.IQueryInterface

METHOD Authenticate : E_AccessLevel
VAR_INPUT
    User   : STRING(32);
    Secret : STRING(32);
END_VAR
END_METHOD

END_INTERFACE

// ---- Interfaces/I_AccessStore.TcIO
// Core §7.7(c) - an access provider whose user table outlives a restart.
// Optional: found by __QUERYINTERFACE on the I_AccessProvider a root was given and
// driven by that root's FB_AccessManager every scan, so a project calls nothing to
// make its users durable. Several roots may share one provider.
INTERFACE I_AccessStore

// Advance the restore, then keep the written table current. TRUE once the
// retained table has been read (or there was none to read).
METHOD M_Service : BOOL
END_METHOD

// TRUE for the rest of this run when the restore found a retained table that was
// corrupt, missing or older than one confirmed written: some users are gone.
METHOD M_RestoreLost : BOOL
END_METHOD

// TRUE while the table on storage is not under control: the latest change could
// not be written (live now, lost at the next restart), or - before M_Service
// returns TRUE - the retained table could not be read.
METHOD M_SaveFailed : BOOL
END_METHOD

END_INTERFACE

// ---- Interfaces/I_HostEventSink.TcIO
// Core §11.6.2 — optional north-bound transport adapter. The publisher and ring
// remain the PLC authority; OPC UA/MES/REST/MQTT implementations only deliver.
INTERFACE I_HostEventSink

METHOD OnHostEvent : BOOL
VAR_IN_OUT
    Ev : ST_HostEvent;
END_VAR
END_METHOD

END_INTERFACE

// ---- Interfaces/I_FieldbusScanner.TcIO
// OPTIONAL Core §10.5.1 / TC3 §10.6 compatibility seam for a deployment that
// needs richer vendor-specific runtime topology discovery. Base Fraktal/TC3 uses
// FB_EcBusHealth + a reviewed project I/O catalog + FB_IoTopologyPublisher; it
// does not require this interface. The fail-closed FB_EcFieldbusScanner skeleton
// is therefore not a default implementation or a base-conformance claim.
// Other buses may implement the same extension without changing the published model.
INTERFACE I_FieldbusScanner

// Rebuild the node table from the master; returns node count (0 = master down).
// Fills Nodes[1..count] (ParentIdx/State/Channels). Called at a slow cadence
// (e.g. 200 ms) — topology changes rarely; live values refresh separately.
METHOD Scan : INT
VAR_IN_OUT
    Data : ST_FieldbusTopology;
END_VAR
END_METHOD

// Update only the live channel values/quality of an already-scanned table (fast
// cadence, every scan). Keeps topology stable while values move.
METHOD RefreshValues : BOOL
VAR_IN_OUT
    Data : ST_FieldbusTopology;
END_VAR
END_METHOD

// Apply/clear an OUTPUT force on one channel (Core §10.5.1, output-only rule).
// MUST already be authorized by the caller (§7.6/§7.7); the scanner only performs
// the write and returns success (FALSE if the channel is an INPUT or unknown).
// Writes the mapped OUTPUT variable through the application — never a raw
// process-image force, never an input, never safety I/O (those are unreachable
// here by construction). Every call is logged by the caller (§8.3).
METHOD ForceChannel : BOOL
VAR_INPUT
    ChannelPath : STRING(255);
    Force       : BOOL;     // TRUE = hold the value, FALSE = release
    BoolValue   : BOOL;     // digital output
    AnalogRaw   : DINT;     // analog output (raw)
END_VAR
END_METHOD

END_INTERFACE

// ---- Interfaces/I_ConfigSource.TcIO
// Core §3.10.2 — a module that contributes entries to the root Unit's
// configuration manifest (static data deliberately excluded from the cyclic
// OPC UA tree and served through the QUERY_CONFIG mailbox instead).
// FB_ModuleBase implements it once for the base-owned facets; composites
// recurse their children, so a new module type inherits participation and
// only overrides M_AppendConfig to add type-owned static data (rare).
// The same walk carries writes back (M_ApplyConfigWrite): read publication
// and write authority stay one participation, so a module cannot end up
// publishing an editable value it has no path to apply (§3.8b).
INTERFACE I_ConfigSource EXTENDS __System.IQueryInterface

// Append this module's (and its children's) manifest entries to the pager.
// Deterministic order across calls — the walk order defines the paging.
METHOD M_AppendConfig : BOOL
VAR_INPUT
    Pager : REFERENCE TO FB_ConfigPager;
END_VAR
END_METHOD

// §3.8d - report what the module named by Scope declared about access to one
// of its registered values. TRUE only from the owner; the root resolves the
// effective level with its policy before it lets a write, capture or set
// record reach the value.
METHOD M_ConfigAccessOf : BOOL
VAR_INPUT
    Scope    : STRING(255);
    WriteKey : STRING(160);
END_VAR
VAR_IN_OUT
    Grant : ST_ConfigAccess;
END_VAR
END_METHOD

// Apply one registered configuration write to the module named by Scope.
// TRUE only from the module that owns the key and accepted the value; a module
// that does not own it returns FALSE so the walk continues past it.
METHOD M_ApplyConfigWrite : BOOL
VAR_INPUT
    Scope     : STRING(255);
    WriteKey  : STRING(160);
    Revision  : UDINT;
    TextValue : STRING(255);
    RootReady : BOOL;
END_VAR
END_METHOD

// §3.8c - capture: store this module's OWN live value into the registered
// field named by WriteKey. No TextValue: the whole point is that the number
// comes from the machine, not from the client. Everything else - revision,
// RequiresReady, the type's own invariants, range, domain, storage - is the
// write path unchanged, so a capture can never accept what a typed write
// would refuse.
METHOD M_ApplyCapture : BOOL
VAR_INPUT
    Scope     : STRING(255);
    WriteKey  : STRING(160);
    Revision  : UDINT;
    RootReady : BOOL;
END_VAR
END_METHOD

// §3.8b — validate one write WITHOUT applying it. Same module, same key lookup,
// same revision check, same RequiresReady rule, same type-specific invariant
// hook, same range and domain checks as M_ApplyConfigWrite — and then nothing
// is stored.
//
// This exists because a parameter-set load is staged and all-or-nothing: every
// record must be proven acceptable BEFORE any value changes, since a
// half-applied machine parametrization is never a valid outcome. A separate
// validation predicate would be free to drift from the write path; this one
// shares the single validator with it, so "would be accepted" and "was
// accepted" cannot disagree.
METHOD M_StageConfigWrite : BOOL
VAR_INPUT
    Scope     : STRING(255);
    WriteKey  : STRING(160);
    Revision  : UDINT;
    TextValue : STRING(255);
    RootReady : BOOL;
END_VAR
END_METHOD

// §3.8b — hand the root ONE not-yet-reported configuration restore loss from
// this module or its children, so the root can annunciate it with the owning
// module's canonical path and apply the deployment's E_ConfigRestorePolicy.
//
// The module marks each loss reported as it hands it over, so the root simply
// drains this until it returns FALSE. That is what makes the annunciation
// exactly-once without either side keeping a list.
METHOD M_TakeRestoreLoss : BOOL
VAR_OUTPUT
    Path     : STRING(80);   // canonical identity of the module that lost it
    Expected : UINT;         // schema version this build understands
    Found    : UINT;         // schema version actually retained
END_VAR
END_METHOD

END_INTERFACE

// ---- Interfaces/I_ConfigPersistence.TcIO
// Core §3.8b — durability of an ACCEPTED write, which is a different question
// from where a parameter SET is stored (I_ConfigStore) and therefore a
// different seam.
//
// §3.8b: "An accepted configuration write shall reach non-volatile storage
// without further operator action, within a declared bounded window." On this
// binding the retentive image is written by the runtime, not by the PLC program,
// so making a value durable is an explicit act with a latency and a failure
// mode - and pretending otherwise is precisely the hope the clause replaces
// with a stated property. FB_UnitBase drives an implementation of this every
// scan and publishes the outcome as PersistPending / PersistFailed.
//
// The shipped default (FB_PersistentDataWriter, LOCAL_RETAIN) needs no wiring:
// a conforming station persists its parametrization with no file system, no
// network and no configuration.
INTERFACE I_ConfigPersistence

// Drive the implementation; called every scan by the owning root. TRUE while a
// durability operation is still in progress, so the root can hold PersistPending
// exactly as long as the value really is not yet safe.
METHOD M_Cyclic : BOOL
END_METHOD

// TRUE when the last completed operation did not make the data durable. Latched
// by the implementation until the next successful one: a failure that clears
// itself before anybody looks is not an answer to "is my configuration safe?".
METHOD M_Failed : BOOL
END_METHOD

// Ask for every write accepted so far to become durable. Returns FALSE if the
// request could not even be started, which is a failure the root publishes
// rather than a silent no-op. Safe to call while one is already in progress.
METHOD M_Request : BOOL
END_METHOD

END_INTERFACE

// ---- Interfaces/I_ConfigStore.TcIO
// Core §3.8b — bounded save / read / list over NAMED parameter sets.
//
// The interface is RECORD-oriented, not document-oriented, and that is the
// whole design. §3.8b forbids a byte image because it carries no per-value
// identity and cannot reject one bad value without rejecting all of them; a
// store that took an opaque blob would reintroduce exactly that one level up.
// Every implementation therefore moves (Scope, WriteKey, ValueType, value)
// records, whatever medium is behind it - retentive memory, a JSON or XML file,
// a database or an MES connector (§3.15).
//
// The store moves records and NOTHING else. It does not validate, does not know
// what a value means, and is never an authorization authority: everything it
// returns is untrusted input, validated on the way in by the owning module's
// typed handler (§5.6, §14).
//
// Save is a three-part transaction - begin, record*, commit - so a half-written
// set never becomes loadable. Read is stateless and addressed by (SetName,
// Index): a cursor would be one more thing to get wrong across a scan boundary.
//
// Queryable: a store that writes its sets out itself (FB_MediumConfigStore) also
// implements I_ConfigPersistence, and the root finds it by __QUERYINTERFACE.
INTERFACE I_ConfigStore EXTENDS __System.IQueryInterface

// How many named sets this store holds, so a client can enumerate them.
METHOD M_Count : INT
END_METHOD

// Remove one named set. FALSE = no set of that name, or a save is open on it
// (a transaction is never pulled from under itself); nothing changed.
METHOD M_Delete : BOOL
VAR_INPUT
    SetName : STRING(80);
END_VAR
END_METHOD

// Header of the Index-th stored set, 1..M_Count, for a bounded listing.
METHOD M_InfoAt : BOOL
VAR_INPUT
    Index : INT;
END_VAR
VAR_IN_OUT
    Info : ST_ConfigSetInfo;
END_VAR
END_METHOD

// Which medium is behind this store - published so an operator can see WHERE
// a saved set actually lives (§3.8b store table).
METHOD M_Kind : E_ConfigStore
END_METHOD

// Header of one stored set. FALSE = no set of that name (Info untouched).
METHOD M_ReadInfo : BOOL
VAR_INPUT
    SetName : STRING(80);
END_VAR
VAR_IN_OUT
    Info : ST_ConfigSetInfo;
END_VAR
END_METHOD

// One record of a stored set, addressed 1..Info.RecordCount. FALSE = absent
// set or out-of-range index (Record untouched).
METHOD M_ReadRecord : BOOL
VAR_INPUT
    SetName : STRING(80);
    Index   : INT;
END_VAR
VAR_IN_OUT
    Record : ST_ConfigRecord;
END_VAR
END_METHOD

// Discard an open save. Always safe to call, including when none is open.
METHOD M_SaveAbort : BOOL
END_METHOD

// Open a save transaction for Info.SetName, overwriting any set of that name
// only when M_SaveCommit succeeds. FALSE = refused (no free slot, empty name,
// a save already open); nothing stored.
METHOD M_SaveBegin : BOOL
VAR_INPUT
    Info : ST_ConfigSetInfo;
END_VAR
END_METHOD

// Close the save and make the set visible to a later read. FALSE = the set was
// not stored; the previous set of that name, if any, is left untouched.
METHOD M_SaveCommit : BOOL
END_METHOD

// Append one record to the open save. FALSE = the set is full or no save is
// open; the transaction is then failed and M_SaveCommit shall refuse it.
METHOD M_SaveRecord : BOOL
VAR_INPUT
    Record : ST_ConfigRecord;
END_VAR
END_METHOD

END_INTERFACE

// ---- Interfaces/I_PersistMedium.TcIO
// Core §3.8b - WHERE retained documents physically live: a file system, the
// controller's retentive memory, a database. Which one is a PROJECT decision, and
// not every platform offers every medium, so the composition root picks one and
// hands the same instance to every consumer; switching medium is that one line.
//
// A medium moves keyed byte documents and nothing else (§3.8b: "the store moves
// bytes"). It validates no content and authorizes nothing: what it returns is
// untrusted input that the consumer validates (§5.6, §14). What it does own is
// the medium's own failure modes - a torn write, a corrupt or vanished copy - so
// a read answers either a whole document it wrote, or that nothing is there, and
// says when a document it confirmed writing is gone (Lost).
//
// Requests are queued and answered asynchronously, because a file or a network
// takes scans; a ticket names one request. The caller's buffer belongs to the
// medium from M_Start* until M_Poll returns TRUE for that ticket. Every caller
// polls its own ticket each scan, and that polling is what advances the medium,
// so a project never schedules it. A zero-length document is a deletion.
INTERFACE I_PersistMedium

// The §3.8b medium class, published by a store built on this medium.
METHOD M_Kind : E_ConfigStore
END_METHOD

// TRUE when a document written here cannot be read back through the
// controller's symbol interfaces (ADS symbols, OPC UA). Only such a medium may
// hold credentials, even salted hashes (§14).
METHOD M_Confidential : BOOL
END_METHOD

// Queue a write of Size bytes at pData under Key (letters, digits, '_', '.',
// '-'; at most 80). 0 = refused: an invalid key or size, or a full queue - ask
// again next scan. The bytes are taken when the write starts, not now.
METHOD M_StartWrite : UDINT
VAR_INPUT
    Key   : STRING(80);
    pData : PVOID;
    Size  : UDINT;
END_VAR
END_METHOD

// Queue a read of the newest valid document under Key into at most Size bytes
// at pData. 0 = refused, as for M_StartWrite.
METHOD M_StartRead : UDINT
VAR_INPUT
    Key   : STRING(80);
    pData : PVOID;
    Size  : UDINT;
END_VAR
END_METHOD

// Advance the medium and report on one ticket. TRUE = that request is finished
// and Result holds its outcome; the ticket is then released. An unknown ticket
// finishes at once with Ok = FALSE, so a caller can never wait forever.
METHOD M_Poll : BOOL
VAR_INPUT
    Ticket : UDINT;
END_VAR
VAR_IN_OUT
    Result : ST_PersistResult;
END_VAR
END_METHOD

END_INTERFACE

